	MoveL Offs(p0,158.4466,180.3462, 0), v100, z5, tool0;
	MoveL Offs(p0,157.43040000000002,179.7648, 0), v100, z5, tool0;
	MoveL Offs(p0,156.14780000000002,179.25060000000002, 0), v100, z5, tool0;
	MoveL Offs(p0,154.6,178.8, 0), v100, z5, tool0;
	MoveL Offs(p0,152.49280000000005,178.35360000000009, 0), v100, z5, tool0;
	MoveL Offs(p0,151.33119999999997,178.07639999999998, 0), v100, z5, tool0;
	MoveL Offs(p0,150.12640000000002,177.77280000000002, 0), v100, z5, tool0;
	MoveL Offs(p0,148.9,177.45, 0), v100, z5, tool0;
	MoveL Offs(p0,147.6736,177.11520000000002, 0), v100, z5, tool0;
	MoveL Offs(p0,146.46880000000002,176.7756, 0), v100, z5, tool0;
	MoveL Offs(p0,145.30720000000002,176.43840000000003, 0), v100, z5, tool0;
	MoveL Offs(p0,144.2104,176.1108, 0), v100, z5, tool0;
	MoveL Offs(p0,143.2,175.8, 0), v100, z5, tool0;
	MoveL Offs(p0,140.56640000000002,175.05440000000004, 0), v100, z5, tool0;
	MoveL Offs(p0,139.6846,174.86759999999998, 0), v100, z5, tool0;
	MoveL Offs(p0,139.0752,174.8272, 0), v100, z5, tool0;
	MoveL Offs(p0,138.725,174.95, 0), v100, z5, tool0;
	MoveL Offs(p0,138.6208,175.25279999999998, 0), v100, z5, tool0;
	MoveL Offs(p0,138.7494,175.7524, 0), v100, z5, tool0;
	MoveL Offs(p0,139.0976,176.46560000000002, 0), v100, z5, tool0;
	MoveL Offs(p0,139.6522,177.4092, 0), v100, z5, tool0;
	MoveL Offs(p0,140.4,178.6, 0), v100, z5, tool0;
	MoveL Offs(p0,142.15320000000003,181.3594, 0), v100, z5, tool0;
	MoveL Offs(p0,142.8384,182.4848, 0), v100, z5, tool0;
	MoveL Offs(p0,143.55,183.675, 0), v100, z5, tool0;
	MoveL Offs(p0,144.27360000000002,184.90720000000002, 0), v100, z5, tool0;
	MoveL Offs(p0,144.9948,186.1586, 0), v100, z5, tool0;
	MoveL Offs(p0,145.69920000000002,187.40640000000002, 0), v100, z5, tool0;
	MoveL Offs(p0,146.37240000000003,188.62780000000004, 0), v100, z5, tool0;
	MoveL Offs(p0,147.0,189.8, 0), v100, z5, tool0;
	MoveL Offs(p0,148.70080000000004,193.01120000000006, 0), v100, z5, tool0;
	MoveL Offs(p0,149.3472,194.0768, 0), v100, z5, tool0;
	MoveL Offs(p0,149.9024,194.80160000000004, 0), v100, z5, tool0;
	MoveL Offs(p0,150.4,195.2, 0), v100, z5, tool0;
	MoveL Offs(p0,150.87359999999998,195.28640000000001, 0), v100, z5, tool0;
	MoveL Offs(p0,151.3568,195.0752, 0), v100, z5, tool0;
	MoveL Offs(p0,151.88320000000002,194.5808, 0), v100, z5, tool0;
	MoveL Offs(p0,152.4864,193.8176, 0), v100, z5, tool0;
	MoveL Offs(p0,153.2,192.8, 0), v100, z5, tool0;
	MoveL Offs(p0,155.14880000000002,190.1568, 0), v100, z5, tool0;
	MoveL Offs(p0,155.675,189.475, 0), v100, z5, tool0;
	MoveL Offs(p0,156.1952,188.8112, 0), v100, z5, tool0;
	MoveL Offs(p0,156.6986,188.17860000000002, 0), v100, z5, tool0;
	MoveL Offs(p0,157.17440000000002,187.5904, 0), v100, z5, tool0;
	MoveL Offs(p0,157.6118,187.0598, 0), v100, z5, tool0;
	MoveL Offs(p0,158.0,186.6, 0), v100, z5, tool0;
	MoveL Offs(p0,158.0,186.6, 0), v100, z5, tool0;
	MoveJ Offs(p0,306.0,172.0, 10), v100, z1, tool0;
	MoveL Offs(p0,305.975,169.764, 0), v100, z5, tool0;
	MoveL Offs(p0,305.89600000000013,167.84000000000006, 0), v100, z5, tool0;
	MoveL Offs(p0,305.757,166.20399999999998, 0), v100, z5, tool0;
	MoveL Offs(p0,305.552,164.83200000000002, 0), v100, z5, tool0;
	MoveL Offs(p0,305.275,163.7, 0), v100, z5, tool0;
	MoveL Offs(p0,304.92,162.784, 0), v100, z5, tool0;
	MoveL Offs(p0,304.48100000000005,162.06, 0), v100, z5, tool0;
	MoveL Offs(p0,303.95200000000006,161.504, 0), v100, z5, tool0;
	MoveL Offs(p0,303.327,161.092, 0), v100, z5, tool0;
	MoveL Offs(p0,302.6,160.8, 0), v100, z5, tool0;
	MoveL Offs(p0,299.23699999999997,159.66620000000003, 0), v100, z5, tool0;
	MoveL Offs(p0,295.4720000000001,158.11360000000008, 0), v100, z5, tool0;
	MoveL Offs(p0,291.431,156.2154, 0), v100, z5, tool0;
	MoveL Offs(p0,287.24000000000007,154.0448, 0), v100, z5, tool0;
	MoveL Offs(p0,283.025,151.675, 0), v100, z5, tool0;
	MoveL Offs(p0,278.912,149.17919999999998, 0), v100, z5, tool0;
	MoveL Offs(p0,275.027,146.6306, 0), v100, z5, tool0;
	MoveL Offs(p0,271.496,144.10240000000002, 0), v100, z5, tool0;
	MoveL Offs(p0,268.44500000000005,141.6678, 0), v100, z5, tool0;
	MoveL Offs(p0,266.0,139.4, 0), v100, z5, tool0;
	MoveL Offs(p0,261.7404,134.63479999999998, 0), v100, z5, tool0;
	MoveL Offs(p0,258.56320000000005,130.29440000000002, 0), v100, z5, tool0;
	MoveL Offs(p0,256.4708,126.37159999999999, 0), v100, z5, tool0;
	MoveL Offs(p0,255.46560000000005,122.85920000000003, 0), v100, z5, tool0;
	MoveL Offs(p0,255.55,119.75, 0), v100, z5, tool0;
	MoveL Offs(p0,256.7264,117.0368, 0), v100, z5, tool0;
	MoveL Offs(p0,258.99719999999996,114.71239999999997, 0), v100, z5, tool0;
	MoveL Offs(p0,262.3648,112.76960000000001, 0), v100, z5, tool0;
	MoveL Offs(p0,266.83160000000004,111.20120000000001, 0), v100, z5, tool0;
	MoveL Offs(p0,272.4,110.0, 0), v100, z5, tool0;
	MoveL Offs(p0,275.49280000000005,109.58740000000003, 0), v100, z5, tool0;
	MoveL Offs(p0,278.59040000000005,109.31520000000005, 0), v100, z5, tool0;
	MoveL Offs(p0,281.7815999999999,109.19179999999999, 0), v100, z5, tool0;
	MoveL Offs(p0,285.15520000000004,109.22560000000001, 0), v100, z5, tool0;
	MoveL Offs(p0,288.8,109.425, 0), v100, z5, tool0;
	MoveL Offs(p0,292.8048,109.79839999999999, 0), v100, z5, tool0;
	MoveL Offs(p0,297.2584,110.35419999999999, 0), v100, z5, tool0;
	MoveL Offs(p0,302.2496,111.10080000000002, 0), v100, z5, tool0;
	MoveL Offs(p0,307.8672,112.04659999999998, 0), v100, z5, tool0;
	MoveL Offs(p0,314.2,113.2, 0), v100, z5, tool0;
	MoveL Offs(p0,317.7136000000001,113.63040000000004, 0), v100, z5, tool0;
	MoveL Offs(p0,319.1914,113.54560000000001, 0), v100, z5, tool0;
	MoveL Offs(p0,320.61280000000005,113.18719999999999, 0), v100, z5, tool0;
	MoveL Offs(p0,322.075,112.5, 0), v100, z5, tool0;
	MoveL Offs(p0,323.6752,111.4288, 0), v100, z5, tool0;
	MoveL Offs(p0,325.5106,109.91839999999999, 0), v100, z5, tool0;
	MoveL Offs(p0,327.67840000000007,107.9136, 0), v100, z5, tool0;
	MoveL Offs(p0,330.2758,105.35920000000002, 0), v100, z5, tool0;
	MoveL Offs(p0,333.4,102.2, 0), v100, z5, tool0;
	MoveL Offs(p0,345.2,90.0, 0), v100, z5, tool0;
	MoveL Offs(p0,335.0,90.0, 0), v100, z5, tool0;
	MoveL Offs(p0,331.073,89.83140000000002, 0), v100, z5, tool0;
	MoveL Offs(p0,326.5760000000001,89.34720000000002, 0), v100, z5, tool0;
	MoveL Offs(p0,321.63499999999993,88.5798, 0), v100, z5, tool0;
	MoveL Offs(p0,316.37600000000003,87.56160000000001, 0), v100, z5, tool0;
	MoveL Offs(p0,310.925,86.325, 0), v100, z5, tool0;
	MoveL Offs(p0,305.408,84.90239999999999, 0), v100, z5, tool0;
	MoveL Offs(p0,299.95099999999996,83.3262, 0), v100, z5, tool0;
	MoveL Offs(p0,294.68,81.6288, 0), v100, z5, tool0;
	MoveL Offs(p0,289.721,79.8426, 0), v100, z5, tool0;
	MoveL Offs(p0,285.2,78.0, 0), v100, z5, tool0;
	MoveL Offs(p0,281.60640000000006,76.04320000000003, 0), v100, z5, tool0;
	MoveL Offs(p0,279.6056,74.80679999999998, 0), v100, z5, tool0;
	MoveL Offs(p0,277.5232,73.43360000000001, 0), v100, z5, tool0;
	MoveL Offs(p0,275.4,71.95, 0), v100, z5, tool0;
	MoveL Offs(p0,273.2768,70.38239999999999, 0), v100, z5, tool0;
	MoveL Offs(p0,271.1944,68.7572, 0), v100, z5, tool0;
	MoveL Offs(p0,269.1936,67.1008, 0), v100, z5, tool0;
	MoveL Offs(p0,267.3152,65.4396, 0), v100, z5, tool0;
	MoveL Offs(p0,265.6,63.8, 0), v100, z5, tool0;
	MoveL Offs(p0,256.0,54.2, 0), v100, z5, tool0;
	MoveL Offs(p0,252.0,62.0, 0), v100, z5, tool0;
	MoveL Offs(p0,249.06160000000006,68.46360000000001, 0), v100, z5, tool0;
	MoveL Offs(p0,246.61280000000005,75.40480000000002, 0), v100, z5, tool0;
	MoveL Offs(p0,244.66319999999996,82.6892, 0), v100, z5, tool0;
	MoveL Offs(p0,243.22240000000002,90.1824, 0), v100, z5, tool0;
	MoveL Offs(p0,242.3,97.75, 0), v100, z5, tool0;
	MoveL Offs(p0,241.9056,105.2576, 0), v100, z5, tool0;
	MoveL Offs(p0,242.04879999999997,112.5708, 0), v100, z5, tool0;
	MoveL Offs(p0,242.73920000000004,119.55520000000001, 0), v100, z5, tool0;
	MoveL Offs(p0,243.9864,126.0764, 0), v100, z5, tool0;
	MoveL Offs(p0,245.8,132.0, 0), v100, z5, tool0;
	MoveL Offs(p0,247.3344000000001,135.71680000000003, 0), v100, z5, tool0;
	MoveL Offs(p0,248.23359999999997,137.6952, 0), v100, z5, tool0;
	MoveL Offs(p0,249.19520000000003,139.70239999999998, 0), v100, z5, tool0;
	MoveL Offs(p0,250.2,141.7, 0), v100, z5, tool0;
	MoveL Offs(p0,251.2288,143.64960000000002, 0), v100, z5, tool0;
	MoveL Offs(p0,252.26239999999999,145.51280000000003, 0), v100, z5, tool0;
	MoveL Offs(p0,253.28160000000003,147.2512, 0), v100, z5, tool0;
	MoveL Offs(p0,254.2672,148.8264, 0), v100, z5, tool0;
	MoveL Offs(p0,255.2,150.2, 0), v100, z5, tool0;
	MoveL Offs(p0,258.3632,154.18440000000004, 0), v100, z5, tool0;
	MoveL Offs(p0,262.43360000000007,158.36320000000006, 0), v100, z5, tool0;
	MoveL Offs(p0,267.2024,162.59480000000002, 0), v100, z5, tool0;
	MoveL Offs(p0,272.46080000000006,166.73760000000001, 0), v100, z5, tool0;
	MoveL Offs(p0,278.0,170.65, 0), v100, z5, tool0;
	MoveL Offs(p0,283.6112,174.1904, 0), v100, z5, tool0;
	MoveL Offs(p0,289.0856,177.2172, 0), v100, z5, tool0;
	MoveL Offs(p0,294.2144,179.58880000000002, 0), v100, z5, tool0;
	MoveL Offs(p0,298.7888,181.1636, 0), v100, z5, tool0;
	MoveL Offs(p0,302.6,181.8, 0), v100, z5, tool0;
	MoveL Offs(p0,305.00640000000004,180.79840000000002, 0), v100, z5, tool0;
	MoveL Offs(p0,305.35,180.05, 0), v100, z5, tool0;
	MoveL Offs(p0,305.6096,179.0496, 0), v100, z5, tool0;
	MoveL Offs(p0,305.7948,177.7708, 0), v100, z5, tool0;
	MoveL Offs(p0,305.9152,176.18720000000002, 0), v100, z5, tool0;
	MoveL Offs(p0,305.98040000000003,174.2724, 0), v100, z5, tool0;
	MoveL Offs(p0,306.0,172.0, 0), v100, z5, tool0;
	MoveL Offs(p0,306.0,172.0, 0), v100, z5, tool0;
	MoveJ Offs(p0,510.0,155.6, 10), v100, z1, tool0;
	MoveL Offs(p0,507.53460000000007,145.5334, 0), v100, z5, tool0;
	MoveL Offs(p0,504.22080000000017,136.09920000000005, 0), v100, z5, tool0;
	MoveL Offs(p0,500.06219999999996,127.30579999999998, 0), v100, z5, tool0;
	MoveL Offs(p0,495.06239999999997,119.16160000000002, 0), v100, z5, tool0;
	MoveL Offs(p0,489.225,111.675, 0), v100, z5, tool0;
	MoveL Offs(p0,482.5536,104.85439999999998, 0), v100, z5, tool0;
	MoveL Offs(p0,475.0517999999999,98.7082, 0), v100, z5, tool0;
	MoveL Offs(p0,466.7232,93.24480000000001, 0), v100, z5, tool0;
	MoveL Offs(p0,457.5714,88.4726, 0), v100, z5, tool0;
	MoveL Offs(p0,447.6,84.4, 0), v100, z5, tool0;
	MoveL Offs(p0,443.93160000000006,83.08260000000001, 0), v100, z5, tool0;
	MoveL Offs(p0,440.62080000000014,81.99680000000002, 0), v100, z5, tool0;
	MoveL Offs(p0,437.50919999999996,81.12219999999999, 0), v100, z5, tool0;
	MoveL Offs(p0,434.4384,80.43839999999999, 0), v100, z5, tool0;
	MoveL Offs(p0,431.25,79.925, 0), v100, z5, tool0;
	MoveL Offs(p0,427.7856,79.5616, 0), v100, z5, tool0;
	MoveL Offs(p0,423.88680000000005,79.3278, 0), v100, z5, tool0;
	MoveL Offs(p0,419.39520000000005,79.20320000000001, 0), v100, z5, tool0;
	MoveL Offs(p0,414.15240000000006,79.1674, 0), v100, z5, tool0;
	MoveL Offs(p0,408.0,79.2, 0), v100, z5, tool0;
	MoveL Offs(p0,398.902,79.31840000000001, 0), v100, z5, tool0;
	MoveL Offs(p0,390.9920000000001,79.69120000000002, 0), v100, z5, tool0;
	MoveL Offs(p0,384.186,80.34479999999999, 0), v100, z5, tool0;
	MoveL Offs(p0,378.4,81.3056, 0), v100, z5, tool0;
	MoveL Offs(p0,373.55,82.6, 0), v100, z5, tool0;
	MoveL Offs(p0,369.552,84.2544, 0), v100, z5, tool0;
	MoveL Offs(p0,366.322,86.2952, 0), v100, z5, tool0;
	MoveL Offs(p0,363.776,88.7488, 0), v100, z5, tool0;
	MoveL Offs(p0,361.83000000000004,91.64160000000001, 0), v100, z5, tool0;
	MoveL Offs(p0,360.4,95.0, 0), v100, z5, tool0;
	MoveL Offs(p0,359.1992000000001,100.0506, 0), v100, z5, tool0;
	MoveL Offs(p0,358.80960000000016,105.52480000000003, 0), v100, z5, tool0;
	MoveL Offs(p0,359.1904,111.30619999999999, 0), v100, z5, tool0;
	MoveL Offs(p0,360.3008000000001,117.2784, 0), v100, z5, tool0;
	MoveL Offs(p0,362.1,123.325, 0), v100, z5, tool0;
	MoveL Offs(p0,364.5472,129.32959999999997, 0), v100, z5, tool0;
	MoveL Offs(p0,367.60159999999996,135.17579999999998, 0), v100, z5, tool0;
	MoveL Offs(p0,371.2224,140.74720000000002, 0), v100, z5, tool0;
	MoveL Offs(p0,375.3688,145.9274, 0), v100, z5, tool0;
	MoveL Offs(p0,380.0,150.6, 0), v100, z5, tool0;
	MoveL Offs(p0,383.889,153.90980000000002, 0), v100, z5, tool0;
	MoveL Offs(p0,387.5680000000001,156.65440000000007, 0), v100, z5, tool0;
	MoveL Offs(p0,391.115,158.8566, 0), v100, z5, tool0;
	MoveL Offs(p0,394.60800000000006,160.5392, 0), v100, z5, tool0;
	MoveL Offs(p0,398.125,161.725, 0), v100, z5, tool0;
	MoveL Offs(p0,401.74399999999997,162.4368, 0), v100, z5, tool0;
	MoveL Offs(p0,405.543,162.69740000000002, 0), v100, z5, tool0;
	MoveL Offs(p0,409.6,162.52960000000002, 0), v100, z5, tool0;
	MoveL Offs(p0,413.99300000000005,161.9562, 0), v100, z5, tool0;
	MoveL Offs(p0,418.8,161.0, 0), v100, z5, tool0;
	MoveL Offs(p0,427.9466000000001,159.2384, 0), v100, z5, tool0;
	MoveL Offs(p0,437.39680000000016,158.13920000000002, 0), v100, z5, tool0;
	MoveL Offs(p0,446.98619999999994,157.6808, 0), v100, z5, tool0;
	MoveL Offs(p0,456.55039999999997,157.8416, 0), v100, z5, tool0;
	MoveL Offs(p0,465.925,158.6, 0), v100, z5, tool0;
	MoveL Offs(p0,474.9456,159.9344, 0), v100, z5, tool0;
	MoveL Offs(p0,483.4477999999999,161.82319999999999, 0), v100, z5, tool0;
	MoveL Offs(p0,491.26720000000006,164.2448, 0), v100, z5, tool0;
	MoveL Offs(p0,498.23940000000005,167.1776, 0), v100, z5, tool0;
	MoveL Offs(p0,504.2,170.6, 0), v100, z5, tool0;
	MoveL Offs(p0,507.44640000000015,172.81280000000004, 0), v100, z5, tool0;
	MoveL Offs(p0,508.5956,173.51420000000002, 0), v100, z5, tool0;
	MoveL Offs(p0,509.4832,173.9504, 0), v100, z5, tool0;
	MoveL Offs(p0,510.15,174.125, 0), v100, z5, tool0;
	MoveL Offs(p0,510.63680000000005,174.0416, 0), v100, z5, tool0;
	MoveL Offs(p0,510.9844,173.7038, 0), v100, z5, tool0;
	MoveL Offs(p0,511.23360000000014,173.11520000000002, 0), v100, z5, tool0;
	MoveL Offs(p0,511.4252,172.2794, 0), v100, z5, tool0;
	MoveL Offs(p0,511.6,171.2, 0), v100, z5, tool0;
	MoveL Offs(p0,511.69539999999995,168.0698, 0), v100, z5, tool0;
	MoveL Offs(p0,511.61280000000005,166.60160000000002, 0), v100, z5, tool0;
	MoveL Offs(p0,511.475,164.975, 0), v100, z5, tool0;
	MoveL Offs(p0,511.28319999999997,163.2224, 0), v100, z5, tool0;
	MoveL Offs(p0,511.0386,161.37619999999998, 0), v100, z5, tool0;
	MoveL Offs(p0,510.7424000000001,159.46880000000002, 0), v100, z5, tool0;
	MoveL Offs(p0,510.39580000000007,157.5326, 0), v100, z5, tool0;
	MoveL Offs(p0,510.0,155.6, 0), v100, z5, tool0;
	MoveL Offs(p0,510.0,155.6, 0), v100, z5, tool0;
	MoveJ Offs(p0,181.4,171.0, 10), v100, z1, tool0;
	MoveL Offs(p0,184.04000000000008,170.41920000000005, 0), v100, z5, tool0;
	MoveL Offs(p0,185.57599999999996,169.9848, 0), v100, z5, tool0;
	MoveL Offs(p0,187.208,169.4736, 0), v100, z5, tool0;
	MoveL Offs(p0,188.9,168.9, 0), v100, z5, tool0;
	MoveL Offs(p0,190.616,168.27839999999998, 0), v100, z5, tool0;
	MoveL Offs(p0,192.32,167.6232, 0), v100, z5, tool0;
	MoveL Offs(p0,193.97600000000003,166.9488, 0), v100, z5, tool0;
	MoveL Offs(p0,195.548,166.26960000000003, 0), v100, z5, tool0;
	MoveL Offs(p0,197.0,165.6, 0), v100, z5, tool0;
	MoveL Offs(p0,205.6,161.4, 0), v100, z5, tool0;
	MoveL Offs(p0,194.4,154.6, 0), v100, z5, tool0;
	MoveL Offs(p0,191.1044,152.5704, 0), v100, z5, tool0;
	MoveL Offs(p0,187.83520000000004,150.33920000000003, 0), v100, z5, tool0;
	MoveL Offs(p0,184.6188,147.9328, 0), v100, z5, tool0;
	MoveL Offs(p0,181.48160000000001,145.3776, 0), v100, z5, tool0;
	MoveL Offs(p0,178.45,142.7, 0), v100, z5, tool0;
	MoveL Offs(p0,175.5504,139.92639999999997, 0), v100, z5, tool0;
	MoveL Offs(p0,172.80919999999998,137.08319999999998, 0), v100, z5, tool0;
	MoveL Offs(p0,170.2528,134.1968, 0), v100, z5, tool0;
	MoveL Offs(p0,167.90760000000003,131.29360000000003, 0), v100, z5, tool0;
	MoveL Offs(p0,165.8,128.4, 0), v100, z5, tool0;
	MoveL Offs(p0,164.20960000000002,126.35360000000003, 0), v100, z5, tool0;
	MoveL Offs(p0,163.4834,125.67839999999998, 0), v100, z5, tool0;
	MoveL Offs(p0,162.72480000000002,125.2288, 0), v100, z5, tool0;
	MoveL Offs(p0,161.875,125.0, 0), v100, z5, tool0;
	MoveL Offs(p0,160.8752,124.98719999999999, 0), v100, z5, tool0;
	MoveL Offs(p0,159.6666,125.1856, 0), v100, z5, tool0;
	MoveL Offs(p0,158.1904,125.5904, 0), v100, z5, tool0;
	MoveL Offs(p0,156.38780000000003,126.19680000000001, 0), v100, z5, tool0;
	MoveL Offs(p0,154.2,127.0, 0), v100, z5, tool0;
	MoveL Offs(p0,150.75400000000002,128.0432, 0), v100, z5, tool0;
	MoveL Offs(p0,146.98400000000004,128.88960000000003, 0), v100, z5, tool0;
	MoveL Offs(p0,143.022,129.53439999999998, 0), v100, z5, tool0;
	MoveL Offs(p0,139.0,129.9728, 0), v100, z5, tool0;
	MoveL Offs(p0,135.05,130.2, 0), v100, z5, tool0;
	MoveL Offs(p0,131.304,130.21120000000002, 0), v100, z5, tool0;
	MoveL Offs(p0,127.894,130.0016, 0), v100, z5, tool0;
	MoveL Offs(p0,124.952,129.56640000000002, 0), v100, z5, tool0;
	MoveL Offs(p0,122.61000000000001,128.9008, 0), v100, z5, tool0;
	MoveL Offs(p0,121.0,128.0, 0), v100, z5, tool0;
	MoveL Offs(p0,119.25280000000002,125.62240000000001, 0), v100, z5, tool0;
	MoveL Offs(p0,118.9,124.875, 0), v100, z5, tool0;
	MoveL Offs(p0,118.5952,124.09759999999999, 0), v100, z5, tool0;
	MoveL Offs(p0,118.34560000000002,123.3058, 0), v100, z5, tool0;
	MoveL Offs(p0,118.15840000000003,122.51520000000001, 0), v100, z5, tool0;
	MoveL Offs(p0,118.04080000000002,121.74140000000003, 0), v100, z5, tool0;
	MoveL Offs(p0,118.0,121.0, 0), v100, z5, tool0;
	MoveL Offs(p0,118.41600000000001,118.59380000000002, 0), v100, z5, tool0;
	MoveL Offs(p0,119.60000000000002,115.7664, 0), v100, z5, tool0;
	MoveL Offs(p0,121.45599999999999,112.62460000000002, 0), v100, z5, tool0;
	MoveL Offs(p0,123.888,109.27520000000001, 0), v100, z5, tool0;
	MoveL Offs(p0,126.8,105.825, 0), v100, z5, tool0;
	MoveL Offs(p0,130.096,102.3808, 0), v100, z5, tool0;
	MoveL Offs(p0,133.68,99.0494, 0), v100, z5, tool0;
	MoveL Offs(p0,137.45600000000002,95.9376, 0), v100, z5, tool0;
	MoveL Offs(p0,141.328,93.15220000000002, 0), v100, z5, tool0;
	MoveL Offs(p0,145.2,90.8, 0), v100, z5, tool0;
	MoveL Offs(p0,148.10080000000005,89.01280000000003, 0), v100, z5, tool0;
	MoveL Offs(p0,149.1672,88.12519999999999, 0), v100, z5, tool0;
	MoveL Offs(p0,150.0224,87.1584, 0), v100, z5, tool0;
	MoveL Offs(p0,150.7,86.05, 0), v100, z5, tool0;
	MoveL Offs(p0,151.2336,84.7376, 0), v100, z5, tool0;
	MoveL Offs(p0,151.6568,83.1588, 0), v100, z5, tool0;
	MoveL Offs(p0,152.00320000000002,81.25120000000001, 0), v100, z5, tool0;
	MoveL Offs(p0,152.3064,78.9524, 0), v100, z5, tool0;
	MoveL Offs(p0,152.6,76.2, 0), v100, z5, tool0;
	MoveL Offs(p0,153.02400000000006,72.40480000000002, 0), v100, z5, tool0;
	MoveL Offs(p0,153.27499999999998,70.5012, 0), v100, z5, tool0;
	MoveL Offs(p0,153.544,68.6384, 0), v100, z5, tool0;
	MoveL Offs(p0,153.825,66.85, 0), v100, z5, tool0;
	MoveL Offs(p0,154.11200000000002,65.16959999999999, 0), v100, z5, tool0;
	MoveL Offs(p0,154.399,63.6308, 0), v100, z5, tool0;
	MoveL Offs(p0,154.68,62.2672, 0), v100, z5, tool0;
	MoveL Offs(p0,154.949,61.1124, 0), v100, z5, tool0;
	MoveL Offs(p0,155.2,60.2, 0), v100, z5, tool0;
	MoveL Offs(p0,156.6,55.2, 0), v100, z5, tool0;
	MoveL Offs(p0,150.8,59.2, 0), v100, z5, tool0;
	MoveL Offs(p0,147.62780000000004,61.26780000000001, 0), v100, z5, tool0;
	MoveL Offs(p0,144.26240000000004,63.14240000000002, 0), v100, z5, tool0;
	MoveL Offs(p0,140.7506,64.81060000000001, 0), v100, z5, tool0;
	MoveL Offs(p0,137.13920000000002,66.25919999999999, 0), v100, z5, tool0;
	MoveL Offs(p0,133.475,67.475, 0), v100, z5, tool0;
	MoveL Offs(p0,129.8048,68.44480000000001, 0), v100, z5, tool0;
	MoveL Offs(p0,126.1754,69.1554, 0), v100, z5, tool0;
	MoveL Offs(p0,122.63360000000003,69.59360000000001, 0), v100, z5, tool0;
	MoveL Offs(p0,119.22619999999999,69.7462, 0), v100, z5, tool0;
	MoveL Offs(p0,116.0,69.6, 0), v100, z5, tool0;
	MoveL Offs(p0,106.6,68.6, 0), v100, z5, tool0;
	MoveL Offs(p0,102.0,81.4, 0), v100, z5, tool0;
	MoveL Offs(p0,99.33760000000001,91.1172, 0), v100, z5, tool0;
	MoveL Offs(p0,98.14880000000002,100.96160000000002, 0), v100, z5, tool0;
	MoveL Offs(p0,98.3712,110.77239999999999, 0), v100, z5, tool0;
	MoveL Offs(p0,99.9424,120.38879999999999, 0), v100, z5, tool0;
	MoveL Offs(p0,102.8,129.65, 0), v100, z5, tool0;
	MoveL Offs(p0,106.8816,138.39520000000002, 0), v100, z5, tool0;
	MoveL Offs(p0,112.12480000000001,146.46359999999999, 0), v100, z5, tool0;
	MoveL Offs(p0,118.4672,153.69440000000003, 0), v100, z5, tool0;
	MoveL Offs(p0,125.84639999999999,159.92680000000001, 0), v100, z5, tool0;
	MoveL Offs(p0,134.2,165.0, 0), v100, z5, tool0;
	MoveL Offs(p0,138.71300000000002,167.16060000000002, 0), v100, z5, tool0;
	MoveL Offs(p0,143.16000000000003,168.96480000000003, 0), v100, z5, tool0;
	MoveL Offs(p0,147.583,170.41619999999998, 0), v100, z5, tool0;
	MoveL Offs(p0,152.02400000000003,171.5184, 0), v100, z5, tool0;
	MoveL Offs(p0,156.525,172.275, 0), v100, z5, tool0;
	MoveL Offs(p0,161.128,172.68959999999998, 0), v100, z5, tool0;
	MoveL Offs(p0,165.875,172.76579999999998, 0), v100, z5, tool0;
	MoveL Offs(p0,170.80800000000005,172.5072, 0), v100, z5, tool0;
	MoveL Offs(p0,175.969,171.9174, 0), v100, z5, tool0;
	MoveL Offs(p0,181.4,171.0, 0), v100, z5, tool0;
	MoveL Offs(p0,181.4,171.0, 0), v100, z5, tool0;
	MoveJ Offs(p0,74.6,166.8, 10), v100, z1, tool0;
	MoveL Offs(p0,77.17280000000002,165.32160000000005, 0), v100, z5, tool0;
	MoveL Offs(p0,78.7202,164.32139999999998, 0), v100, z5, tool0;
	MoveL Offs(p0,80.39840000000001,163.18080000000003, 0), v100, z5, tool0;
	MoveL Offs(p0,82.175,161.925, 0), v100, z5, tool0;
	MoveL Offs(p0,84.0176,160.5792, 0), v100, z5, tool0;
	MoveL Offs(p0,85.8938,159.1686, 0), v100, z5, tool0;
	MoveL Offs(p0,87.77120000000001,157.71840000000003, 0), v100, z5, tool0;
	MoveL Offs(p0,89.6174,156.2538, 0), v100, z5, tool0;
	MoveL Offs(p0,91.4,154.8, 0), v100, z5, tool0;
	MoveL Offs(p0,101.6,146.0, 0), v100, z5, tool0;
	MoveL Offs(p0,97.8,136.0, 0), v100, z5, tool0;
	MoveL Offs(p0,96.63680000000002,132.6048, 0), v100, z5, tool0;
	MoveL Offs(p0,96.09719999999999,130.9222, 0), v100, z5, tool0;
	MoveL Offs(p0,95.5984,129.28640000000001, 0), v100, z5, tool0;
	MoveL Offs(p0,95.15,127.725, 0), v100, z5, tool0;
	MoveL Offs(p0,94.7616,126.26559999999999, 0), v100, z5, tool0;
	MoveL Offs(p0,94.4428,124.9358, 0), v100, z5, tool0;
	MoveL Offs(p0,94.20320000000001,123.76320000000001, 0), v100, z5, tool0;
	MoveL Offs(p0,94.0524,122.77540000000002, 0), v100, z5, tool0;
	MoveL Offs(p0,94.0,122.0, 0), v100, z5, tool0;
	MoveL Offs(p0,93.52440000000001,118.99960000000002, 0), v100, z5, tool0;
	MoveL Offs(p0,92.18720000000002,117.48480000000002, 0), v100, z5, tool0;
	MoveL Offs(p0,90.1228,117.34520000000002, 0), v100, z5, tool0;
	MoveL Offs(p0,87.46560000000001,118.4704, 0), v100, z5, tool0;
	MoveL Offs(p0,84.35,120.75, 0), v100, z5, tool0;
	MoveL Offs(p0,80.9104,124.07359999999998, 0), v100, z5, tool0;
	MoveL Offs(p0,77.28119999999998,128.3308, 0), v100, z5, tool0;
	MoveL Offs(p0,73.5968,133.4112, 0), v100, z5, tool0;
	MoveL Offs(p0,69.9916,139.20440000000002, 0), v100, z5, tool0;
	MoveL Offs(p0,66.6,145.6, 0), v100, z5, tool0;
	MoveL Offs(p0,64.8994,149.04300000000003, 0), v100, z5, tool0;
	MoveL Offs(p0,63.50720000000001,151.97600000000006, 0), v100, z5, tool0;
	MoveL Offs(p0,62.407799999999995,154.46499999999997, 0), v100, z5, tool0;
	MoveL Offs(p0,61.5856,156.57600000000002, 0), v100, z5, tool0;
	MoveL Offs(p0,61.025,158.375, 0), v100, z5, tool0;
	MoveL Offs(p0,60.71039999999999,159.92799999999997, 0), v100, z5, tool0;
	MoveL Offs(p0,60.6262,161.30100000000002, 0), v100, z5, tool0;
	MoveL Offs(p0,60.7568,162.56, 0), v100, z5, tool0;
	MoveL Offs(p0,61.0866,163.77100000000002, 0), v100, z5, tool0;
	MoveL Offs(p0,61.6,165.0, 0), v100, z5, tool0;
	MoveL Offs(p0,63.201600000000006,167.83680000000007, 0), v100, z5, tool0;
	MoveL Offs(p0,64.01740000000001,168.7782, 0), v100, z5, tool0;
	MoveL Offs(p0,64.90880000000001,169.40640000000002, 0), v100, z5, tool0;
	MoveL Offs(p0,65.925,169.725, 0), v100, z5, tool0;
	MoveL Offs(p0,67.1152,169.7376, 0), v100, z5, tool0;
	MoveL Offs(p0,68.52860000000001,169.4478, 0), v100, z5, tool0;
	MoveL Offs(p0,70.21440000000001,168.85920000000002, 0), v100, z5, tool0;
	MoveL Offs(p0,72.2218,167.9754, 0), v100, z5, tool0;
	MoveL Offs(p0,74.6,166.8, 0), v100, z5, tool0;
	MoveL Offs(p0,74.6,166.8, 0), v100, z5, tool0;
	MoveJ Offs(p0,247.6,158.2, 10), v100, z1, tool0;
	MoveL Offs(p0,252.2,158.0, 0), v100, z5, tool0;
	MoveL Offs(p0,248.2,152.2, 0), v100, z5, tool0;
	MoveL Offs(p0,246.82720000000012,150.19520000000006, 0), v100, z5, tool0;
	MoveL Offs(p0,246.1228,149.07879999999997, 0), v100, z5, tool0;
	MoveL Offs(p0,245.42560000000003,147.9216, 0), v100, z5, tool0;
	MoveL Offs(p0,244.75,146.75, 0), v100, z5, tool0;
	MoveL Offs(p0,244.11040000000003,145.5904, 0), v100, z5, tool0;
	MoveL Offs(p0,243.5212,144.4692, 0), v100, z5, tool0;
	MoveL Offs(p0,242.99680000000004,143.4128, 0), v100, z5, tool0;
	MoveL Offs(p0,242.5516,142.44760000000002, 0), v100, z5, tool0;
	MoveL Offs(p0,242.2,141.6, 0), v100, z5, tool0;
	MoveL Offs(p0,241.1328000000001,139.28320000000002, 0), v100, z5, tool0;
	MoveL Offs(p0,240.4252,138.4158, 0), v100, z5, tool0;
	MoveL Offs(p0,239.5184,137.7056, 0), v100, z5, tool0;
	MoveL Offs(p0,238.35,137.125, 0), v100, z5, tool0;
	MoveL Offs(p0,236.8576,136.6464, 0), v100, z5, tool0;
	MoveL Offs(p0,234.9788,136.2422, 0), v100, z5, tool0;
	MoveL Offs(p0,232.65120000000007,135.8848, 0), v100, z5, tool0;
	MoveL Offs(p0,229.81239999999997,135.5466, 0), v100, z5, tool0;
	MoveL Offs(p0,226.4,135.2, 0), v100, z5, tool0;
	MoveL Offs(p0,218.27900000000005,133.9028, 0), v100, z5, tool0;
	MoveL Offs(p0,210.36800000000002,131.78240000000002, 0), v100, z5, tool0;
	MoveL Offs(p0,202.865,128.9756, 0), v100, z5, tool0;
	MoveL Offs(p0,195.968,125.61920000000002, 0), v100, z5, tool0;
	MoveL Offs(p0,189.875,121.85, 0), v100, z5, tool0;
	MoveL Offs(p0,184.784,117.8048, 0), v100, z5, tool0;
	MoveL Offs(p0,180.89299999999997,113.62039999999999, 0), v100, z5, tool0;
	MoveL Offs(p0,178.40000000000003,109.4336, 0), v100, z5, tool0;
	MoveL Offs(p0,177.503,105.38119999999999, 0), v100, z5, tool0;
	MoveL Offs(p0,178.4,101.6, 0), v100, z5, tool0;
	MoveL Offs(p0,180.97600000000006,98.31360000000004, 0), v100, z5, tool0;
	MoveL Offs(p0,182.909,96.88040000000001, 0), v100, z5, tool0;
	MoveL Offs(p0,185.32800000000003,95.56480000000002, 0), v100, z5, tool0;
	MoveL Offs(p0,188.275,94.35, 0), v100, z5, tool0;
	MoveL Offs(p0,191.792,93.2192, 0), v100, z5, tool0;
	MoveL Offs(p0,195.921,92.1556, 0), v100, z5, tool0;
	MoveL Offs(p0,200.704,91.14240000000002, 0), v100, z5, tool0;
	MoveL Offs(p0,206.183,90.16279999999999, 0), v100, z5, tool0;
	MoveL Offs(p0,212.4,89.2, 0), v100, z5, tool0;
	MoveL Offs(p0,215.82420000000002,88.67300000000002, 0), v100, z5, tool0;
	MoveL Offs(p0,219.10560000000004,88.17600000000002, 0), v100, z5, tool0;
	MoveL Offs(p0,222.19740000000002,87.71499999999999, 0), v100, z5, tool0;
	MoveL Offs(p0,225.05280000000002,87.296, 0), v100, z5, tool0;
	MoveL Offs(p0,227.625,86.925, 0), v100, z5, tool0;
	MoveL Offs(p0,229.8672,86.608, 0), v100, z5, tool0;
	MoveL Offs(p0,231.7326,86.351, 0), v100, z5, tool0;
	MoveL Offs(p0,233.17440000000002,86.16000000000001, 0), v100, z5, tool0;
	MoveL Offs(p0,234.1458,86.041, 0), v100, z5, tool0;
	MoveL Offs(p0,234.6,86.0, 0), v100, z5, tool0;
	MoveL Offs(p0,235.90240000000003,83.952, 0), v100, z5, tool0;
	MoveL Offs(p0,236.375,82.9, 0), v100, z5, tool0;
	MoveL Offs(p0,236.88959999999997,81.67999999999999, 0), v100, z5, tool0;
	MoveL Offs(p0,237.43779999999998,80.31599999999999, 0), v100, z5, tool0;
	MoveL Offs(p0,238.0112,78.83200000000001, 0), v100, z5, tool0;
	MoveL Offs(p0,238.6014,77.252, 0), v100, z5, tool0;
	MoveL Offs(p0,239.2,75.6, 0), v100, z5, tool0;
	MoveL Offs(p0,240.38080000000005,72.06560000000003, 0), v100, z5, tool0;
	MoveL Offs(p0,241.02519999999998,70.3044, 0), v100, z5, tool0;
	MoveL Offs(p0,241.6864,68.58879999999999, 0), v100, z5, tool0;
	MoveL Offs(p0,242.35,66.95, 0), v100, z5, tool0;
	MoveL Offs(p0,243.00159999999997,65.4192, 0), v100, z5, tool0;
	MoveL Offs(p0,243.62679999999995,64.02759999999999, 0), v100, z5, tool0;
	MoveL Offs(p0,244.21120000000002,62.80640000000001, 0), v100, z5, tool0;
	MoveL Offs(p0,244.74040000000005,61.78679999999999, 0), v100, z5, tool0;
	MoveL Offs(p0,245.2,61.0, 0), v100, z5, tool0;
	MoveL Offs(p0,247.04320000000007,58.04160000000002, 0), v100, z5, tool0;
	MoveL Offs(p0,247.54180000000002,56.9464, 0), v100, z5, tool0;
	MoveL Offs(p0,247.7536,56.100800000000014, 0), v100, z5, tool0;
	MoveL Offs(p0,247.675,55.5, 0), v100, z5, tool0;
	MoveL Offs(p0,247.30239999999998,55.1392, 0), v100, z5, tool0;
	MoveL Offs(p0,246.6322,55.0136, 0), v100, z5, tool0;
	MoveL Offs(p0,245.66080000000002,55.11840000000001, 0), v100, z5, tool0;
	MoveL Offs(p0,244.3846,55.448800000000006, 0), v100, z5, tool0;
	MoveL Offs(p0,242.8,56.0, 0), v100, z5, tool0;
	MoveL Offs(p0,238.1166,57.2124, 0), v100, z5, tool0;
	MoveL Offs(p0,232.18880000000007,57.87520000000002, 0), v100, z5, tool0;
	MoveL Offs(p0,225.32019999999997,58.0268, 0), v100, z5, tool0;
	MoveL Offs(p0,217.81440000000006,57.705600000000004, 0), v100, z5, tool0;
	MoveL Offs(p0,209.975,56.95, 0), v100, z5, tool0;
	MoveL Offs(p0,202.10559999999998,55.798399999999994, 0), v100, z5, tool0;
	MoveL Offs(p0,194.50979999999998,54.28920000000001, 0), v100, z5, tool0;
	MoveL Offs(p0,187.49120000000002,52.46079999999999, 0), v100, z5, tool0;
	MoveL Offs(p0,181.35340000000002,50.351600000000005, 0), v100, z5, tool0;
	MoveL Offs(p0,176.4,48.0, 0), v100, z5, tool0;
	MoveL Offs(p0,174.28800000000007,46.739200000000004, 0), v100, z5, tool0;
	MoveL Offs(p0,173.29500000000002,46.1658, 0), v100, z5, tool0;
	MoveL Offs(p0,172.368,45.641600000000004, 0), v100, z5, tool0;
	MoveL Offs(p0,171.525,45.175, 0), v100, z5, tool0;
	MoveL Offs(p0,170.78400000000002,44.7744, 0), v100, z5, tool0;
	MoveL Offs(p0,170.163,44.4482, 0), v100, z5, tool0;
	MoveL Offs(p0,169.68,44.2048, 0), v100, z5, tool0;
	MoveL Offs(p0,169.353,44.0526, 0), v100, z5, tool0;
	MoveL Offs(p0,169.2,44.0, 0), v100, z5, tool0;
	MoveL Offs(p0,166.80419999999998,48.066199999999995, 0), v100, z5, tool0;
	MoveL Offs(p0,165.7184,50.8224, 0), v100, z5, tool0;
	MoveL Offs(p0,164.575,54.025, 0), v100, z5, tool0;
	MoveL Offs(p0,163.42559999999997,57.5216, 0), v100, z5, tool0;
	MoveL Offs(p0,162.3218,61.159800000000004, 0), v100, z5, tool0;
	MoveL Offs(p0,161.3152,64.78720000000001, 0), v100, z5, tool0;
	MoveL Offs(p0,160.4574,68.25140000000002, 0), v100, z5, tool0;
	MoveL Offs(p0,159.8,71.4, 0), v100, z5, tool0;
	MoveL Offs(p0,159.24020000000002,75.45660000000001, 0), v100, z5, tool0;
	MoveL Offs(p0,158.99360000000004,79.78080000000003, 0), v100, z5, tool0;
	MoveL Offs(p0,159.0494,84.30420000000001, 0), v100, z5, tool0;
	MoveL Offs(p0,159.3968,88.95840000000003, 0), v100, z5, tool0;
	MoveL Offs(p0,160.025,93.675, 0), v100, z5, tool0;
	MoveL Offs(p0,160.9232,98.3856, 0), v100, z5, tool0;
	MoveL Offs(p0,162.0806,103.02179999999998, 0), v100, z5, tool0;
	MoveL Offs(p0,163.4864,107.51520000000001, 0), v100, z5, tool0;
	MoveL Offs(p0,165.1298,111.79740000000001, 0), v100, z5, tool0;
	MoveL Offs(p0,167.0,115.8, 0), v100, z5, tool0;
	MoveL Offs(p0,169.18,119.63700000000001, 0), v100, z5, tool0;
	MoveL Offs(p0,171.93600000000006,123.64800000000002, 0), v100, z5, tool0;
	MoveL Offs(p0,175.17199999999997,127.74299999999998, 0), v100, z5, tool0;
	MoveL Offs(p0,178.792,131.83200000000002, 0), v100, z5, tool0;
	MoveL Offs(p0,182.7,135.825, 0), v100, z5, tool0;
	MoveL Offs(p0,186.8,139.632, 0), v100, z5, tool0;
	MoveL Offs(p0,190.996,143.163, 0), v100, z5, tool0;
	MoveL Offs(p0,195.192,146.32800000000003, 0), v100, z5, tool0;
	MoveL Offs(p0,199.292,149.03699999999998, 0), v100, z5, tool0;
	MoveL Offs(p0,203.2,151.2, 0), v100, z5, tool0;
	MoveL Offs(p0,206.5072,152.7036, 0), v100, z5, tool0;
	MoveL Offs(p0,210.02560000000008,154.08480000000003, 0), v100, z5, tool0;
	MoveL Offs(p0,213.6904,155.32920000000001, 0), v100, z5, tool0;
	MoveL Offs(p0,217.43680000000003,156.42239999999998, 0), v100, z5, tool0;
	MoveL Offs(p0,221.2,157.35, 0), v100, z5, tool0;
	MoveL Offs(p0,224.9152,158.0976, 0), v100, z5, tool0;
	MoveL Offs(p0,228.5176,158.6508, 0), v100, z5, tool0;
	MoveL Offs(p0,231.94240000000005,158.9952, 0), v100, z5, tool0;
	MoveL Offs(p0,235.1248,159.11640000000003, 0), v100, z5, tool0;
	MoveL Offs(p0,238.0,159.0, 0), v100, z5, tool0;
	MoveL Offs(p0,240.817,158.68859999999998, 0), v100, z5, tool0;
	MoveL Offs(p0,241.84,158.60320000000002, 0), v100, z5, tool0;
	MoveL Offs(p0,242.875,158.525, 0), v100, z5, tool0;
	MoveL Offs(p0,243.904,158.4528, 0), v100, z5, tool0;
	MoveL Offs(p0,244.90900000000002,158.38539999999998, 0), v100, z5, tool0;
	MoveL Offs(p0,245.872,158.32160000000002, 0), v100, z5, tool0;
	MoveL Offs(p0,246.775,158.2602, 0), v100, z5, tool0;
	MoveL Offs(p0,247.6,158.2, 0), v100, z5, tool0;
	MoveL Offs(p0,247.6,158.2, 0), v100, z5, tool0;
	MoveJ Offs(p0,316.6,127.2, 10), v100, z1, tool0;
	MoveL Offs(p0,317.69760000000014,124.67520000000002, 0), v100, z5, tool0;
	MoveL Offs(p0,318.1624,123.52079999999998, 0), v100, z5, tool0;
	MoveL Offs(p0,318.5648,122.4576, 0), v100, z5, tool0;
	MoveL Offs(p0,318.9,121.5, 0), v100, z5, tool0;
	MoveL Offs(p0,319.1632,120.6624, 0), v100, z5, tool0;
	MoveL Offs(p0,319.3496,119.95920000000001, 0), v100, z5, tool0;
	MoveL Offs(p0,319.4544,119.40480000000002, 0), v100, z5, tool0;
	MoveL Offs(p0,319.4728,119.0136, 0), v100, z5, tool0;
	MoveL Offs(p0,319.4,118.8, 0), v100, z5, tool0;
	MoveL Offs(p0,315.29600000000005,117.70880000000004, 0), v100, z5, tool0;
	MoveL Offs(p0,311.183,116.89020000000001, 0), v100, z5, tool0;
	MoveL Offs(p0,306.2,115.97440000000002, 0), v100, z5, tool0;
	MoveL Offs(p0,300.725,115.025, 0), v100, z5, tool0;
	MoveL Offs(p0,295.13599999999997,114.10559999999998, 0), v100, z5, tool0;
	MoveL Offs(p0,289.811,113.2798, 0), v100, z5, tool0;
	MoveL Offs(p0,285.12800000000004,112.61120000000001, 0), v100, z5, tool0;
	MoveL Offs(p0,281.46500000000003,112.1634, 0), v100, z5, tool0;
	MoveL Offs(p0,279.2,112.0, 0), v100, z5, tool0;
	MoveL Offs(p0,276.77700000000004,112.1152, 0), v100, z5, tool0;
	MoveL Offs(p0,274.24000000000007,112.44160000000004, 0), v100, z5, tool0;
	MoveL Offs(p0,271.667,112.95039999999999, 0), v100, z5, tool0;
	MoveL Offs(p0,269.136,113.61280000000002, 0), v100, z5, tool0;
	MoveL Offs(p0,266.725,114.4, 0), v100, z5, tool0;
	MoveL Offs(p0,264.512,115.28320000000001, 0), v100, z5, tool0;
	MoveL Offs(p0,262.575,116.2336, 0), v100, z5, tool0;
	MoveL Offs(p0,260.992,117.22240000000002, 0), v100, z5, tool0;
	MoveL Offs(p0,259.841,118.22080000000001, 0), v100, z5, tool0;
	MoveL Offs(p0,259.2,119.2, 0), v100, z5, tool0;
	MoveL Offs(p0,258.98260000000005,122.45520000000002, 0), v100, z5, tool0;
	MoveL Offs(p0,260.34080000000006,126.32960000000006, 0), v100, z5, tool0;
	MoveL Offs(p0,263.0502,130.62640000000002, 0), v100, z5, tool0;
	MoveL Offs(p0,266.8864,135.1488, 0), v100, z5, tool0;
	MoveL Offs(p0,271.625,139.7, 0), v100, z5, tool0;
	MoveL Offs(p0,277.0416,144.08319999999998, 0), v100, z5, tool0;
	MoveL Offs(p0,282.9118,148.10160000000002, 0), v100, z5, tool0;
	MoveL Offs(p0,289.01120000000003,151.55840000000003, 0), v100, z5, tool0;
	MoveL Offs(p0,295.1154,154.25680000000003, 0), v100, z5, tool0;
	MoveL Offs(p0,301.0,156.0, 0), v100, z5, tool0;
	MoveL Offs(p0,303.8768000000001,156.47680000000005, 0), v100, z5, tool0;
	MoveL Offs(p0,304.94019999999995,156.44819999999999, 0), v100, z5, tool0;
	MoveL Offs(p0,305.8224,156.1664, 0), v100, z5, tool0;
	MoveL Offs(p0,306.575,155.575, 0), v100, z5, tool0;
	MoveL Offs(p0,307.2496,154.61759999999998, 0), v100, z5, tool0;
	MoveL Offs(p0,307.8978,153.23780000000002, 0), v100, z5, tool0;
	MoveL Offs(p0,308.57120000000003,151.37920000000003, 0), v100, z5, tool0;
	MoveL Offs(p0,309.3214,148.9854, 0), v100, z5, tool0;
	MoveL Offs(p0,310.2,146.0, 0), v100, z5, tool0;
	MoveL Offs(p0,311.3840000000001,142.14400000000003, 0), v100, z5, tool0;
	MoveL Offs(p0,312.036,140.087, 0), v100, z5, tool0;
	MoveL Offs(p0,312.71200000000005,138.0, 0), v100, z5, tool0;
	MoveL Offs(p0,313.4,135.925, 0), v100, z5, tool0;
	MoveL Offs(p0,314.08799999999997,133.904, 0), v100, z5, tool0;
	MoveL Offs(p0,314.764,131.97899999999998, 0), v100, z5, tool0;
	MoveL Offs(p0,315.41600000000005,130.192, 0), v100, z5, tool0;
	MoveL Offs(p0,316.03200000000004,128.585, 0), v100, z5, tool0;
	MoveL Offs(p0,316.6,127.2, 0), v100, z5, tool0;
	MoveL Offs(p0,316.6,127.2, 0), v100, z5, tool0;
	MoveJ Offs(p0,236.8,132.8, 10), v100, z1, tool0;
	MoveL Offs(p0,238.77280000000002,130.28, 0), v100, z5, tool0;
	MoveL Offs(p0,238.7054,129.552, 0), v100, z5, tool0;
	MoveL Offs(p0,238.52160000000003,128.704, 0), v100, z5, tool0;
	MoveL Offs(p0,238.22020000000003,127.724, 0), v100, z5, tool0;
	MoveL Offs(p0,237.8,126.6, 0), v100, z5, tool0;
	MoveL Offs(p0,237.22880000000004,124.26240000000004, 0), v100, z5, tool0;
	MoveL Offs(p0,236.97020000000003,122.5806, 0), v100, z5, tool0;
	MoveL Offs(p0,236.7344,120.6192, 0), v100, z5, tool0;
	MoveL Offs(p0,236.525,118.425, 0), v100, z5, tool0;
	MoveL Offs(p0,236.34560000000002,116.04479999999998, 0), v100, z5, tool0;
	MoveL Offs(p0,236.1998,113.52539999999999, 0), v100, z5, tool0;
	MoveL Offs(p0,236.09120000000001,110.9136, 0), v100, z5, tool0;
	MoveL Offs(p0,236.02340000000004,108.25619999999999, 0), v100, z5, tool0;
	MoveL Offs(p0,236.0,105.6, 0), v100, z5, tool0;
	MoveL Offs(p0,236.0,89.6, 0), v100, z5, tool0;
	MoveL Offs(p0,229.6,90.6, 0), v100, z5, tool0;
	MoveL Offs(p0,226.9168000000001,91.02240000000003, 0), v100, z5, tool0;
	MoveL Offs(p0,225.24219999999997,91.2696, 0), v100, z5, tool0;
	MoveL Offs(p0,223.39840000000004,91.53120000000001, 0), v100, z5, tool0;
	MoveL Offs(p0,221.425,91.8, 0), v100, z5, tool0;
	MoveL Offs(p0,219.3616,92.06880000000001, 0), v100, z5, tool0;
	MoveL Offs(p0,217.2478,92.33039999999998, 0), v100, z5, tool0;
	MoveL Offs(p0,215.1232,92.5776, 0), v100, z5, tool0;
	MoveL Offs(p0,213.02740000000003,92.80320000000002, 0), v100, z5, tool0;
	MoveL Offs(p0,211.0,93.0, 0), v100, z5, tool0;
	MoveL Offs(p0,201.3376,94.36460000000002, 0), v100, z5, tool0;
	MoveL Offs(p0,193.48480000000004,96.26080000000003, 0), v100, z5, tool0;
	MoveL Offs(p0,187.46319999999997,98.6322, 0), v100, z5, tool0;
	MoveL Offs(p0,183.29440000000005,101.4224, 0), v100, z5, tool0;
	MoveL Offs(p0,181.0,104.575, 0), v100, z5, tool0;
	MoveL Offs(p0,180.60160000000002,108.0336, 0), v100, z5, tool0;
	MoveL Offs(p0,182.1208,111.74180000000001, 0), v100, z5, tool0;
	MoveL Offs(p0,185.57920000000001,115.64320000000002, 0), v100, z5, tool0;
	MoveL Offs(p0,190.9984,119.68140000000001, 0), v100, z5, tool0;
	MoveL Offs(p0,198.4,123.8, 0), v100, z5, tool0;
	MoveL Offs(p0,200.57080000000002,124.8232, 0), v100, z5, tool0;
	MoveL Offs(p0,202.85440000000003,125.84160000000004, 0), v100, z5, tool0;
	MoveL Offs(p0,205.2076,126.83840000000001, 0), v100, z5, tool0;
	MoveL Offs(p0,207.58720000000002,127.7968, 0), v100, z5, tool0;
	MoveL Offs(p0,209.95,128.7, 0), v100, z5, tool0;
	MoveL Offs(p0,212.25279999999998,129.5312, 0), v100, z5, tool0;
	MoveL Offs(p0,214.45239999999998,130.2736, 0), v100, z5, tool0;
	MoveL Offs(p0,216.50560000000004,130.9104, 0), v100, z5, tool0;
	MoveL Offs(p0,218.3692,131.4248, 0), v100, z5, tool0;
	MoveL Offs(p0,220.0,131.8, 0), v100, z5, tool0;
	MoveL Offs(p0,223.2406,132.449, 0), v100, z5, tool0;
	MoveL Offs(p0,225.9328000000001,132.96000000000004, 0), v100, z5, tool0;
	MoveL Offs(p0,228.1522,133.339, 0), v100, z5, tool0;
	MoveL Offs(p0,229.9744,133.592, 0), v100, z5, tool0;
	MoveL Offs(p0,231.475,133.725, 0), v100, z5, tool0;
	MoveL Offs(p0,232.72960000000003,133.744, 0), v100, z5, tool0;
	MoveL Offs(p0,233.8138,133.655, 0), v100, z5, tool0;
	MoveL Offs(p0,234.8032,133.464, 0), v100, z5, tool0;
	MoveL Offs(p0,235.77339999999998,133.177, 0), v100, z5, tool0;
	MoveL Offs(p0,236.8,132.8, 0), v100, z5, tool0;
	MoveL Offs(p0,236.8,132.8, 0), v100, z5, tool0;
	MoveJ Offs(p0,154.4,123.4, 10), v100, z1, tool0;
	MoveL Offs(p0,161.8,120.4, 0), v100, z5, tool0;
	MoveL Offs(p0,157.8,110.2, 0), v100, z5, tool0;
	MoveL Offs(p0,156.63680000000002,106.78400000000003, 0), v100, z5, tool0;
	MoveL Offs(p0,156.0972,105.079, 0), v100, z5, tool0;
	MoveL Offs(p0,155.5984,103.41600000000001, 0), v100, z5, tool0;
	MoveL Offs(p0,155.15,101.825, 0), v100, z5, tool0;
	MoveL Offs(p0,154.7616,100.336, 0), v100, z5, tool0;
	MoveL Offs(p0,154.44279999999998,98.979, 0), v100, z5, tool0;
	MoveL Offs(p0,154.2032,97.784, 0), v100, z5, tool0;
	MoveL Offs(p0,154.05239999999998,96.78100000000002, 0), v100, z5, tool0;
	MoveL Offs(p0,154.0,96.0, 0), v100, z5, tool0;
	MoveL Offs(p0,153.55040000000002,93.45760000000003, 0), v100, z5, tool0;
	MoveL Offs(p0,152.96859999999998,92.7114, 0), v100, z5, tool0;
	MoveL Offs(p0,152.1312,92.3168, 0), v100, z5, tool0;
	MoveL Offs(p0,151.025,92.275, 0), v100, z5, tool0;
	MoveL Offs(p0,149.6368,92.5872, 0), v100, z5, tool0;
	MoveL Offs(p0,147.95340000000002,93.25460000000001, 0), v100, z5, tool0;
	MoveL Offs(p0,145.96160000000003,94.2784, 0), v100, z5, tool0;
	MoveL Offs(p0,143.6482,95.65979999999999, 0), v100, z5, tool0;
	MoveL Offs(p0,141.0,97.4, 0), v100, z5, tool0;
	MoveL Offs(p0,136.74640000000002,100.4204, 0), v100, z5, tool0;
	MoveL Offs(p0,132.89120000000003,103.56320000000002, 0), v100, z5, tool0;
	MoveL Offs(p0,129.4728,106.77080000000001, 0), v100, z5, tool0;
	MoveL Offs(p0,126.5296,109.9856, 0), v100, z5, tool0;
	MoveL Offs(p0,124.1,113.15, 0), v100, z5, tool0;
	MoveL Offs(p0,122.2224,116.2064, 0), v100, z5, tool0;
	MoveL Offs(p0,120.93519999999998,119.09720000000002, 0), v100, z5, tool0;
	MoveL Offs(p0,120.27680000000001,121.76480000000001, 0), v100, z5, tool0;
	MoveL Offs(p0,120.28560000000002,124.1516, 0), v100, z5, tool0;
	MoveL Offs(p0,121.0,126.2, 0), v100, z5, tool0;
	MoveL Offs(p0,124.30080000000002,127.46400000000006, 0), v100, z5, tool0;
	MoveL Offs(p0,127.2442,127.71199999999999, 0), v100, z5, tool0;
	MoveL Offs(p0,130.79840000000002,127.72000000000003, 0), v100, z5, tool0;
	MoveL Offs(p0,134.775,127.5, 0), v100, z5, tool0;
	MoveL Offs(p0,138.9856,127.064, 0), v100, z5, tool0;
	MoveL Offs(p0,143.2418,126.424, 0), v100, z5, tool0;
	MoveL Offs(p0,147.35520000000002,125.59200000000001, 0), v100, z5, tool0;
	MoveL Offs(p0,151.1374,124.58000000000001, 0), v100, z5, tool0;
	MoveL Offs(p0,154.4,123.4, 0), v100, z5, tool0;
	MoveL Offs(p0,154.4,123.4, 0), v100, z5, tool0;
	MoveJ Offs(p0,368.6,80.0, 10), v100, z1, tool0;
	MoveL Offs(p0,374.8776000000001,77.93640000000002, 0), v100, z5, tool0;
	MoveL Offs(p0,381.21280000000013,76.18720000000003, 0), v100, z5, tool0;
	MoveL Offs(p0,387.5792,74.7548, 0), v100, z5, tool0;
	MoveL Offs(p0,393.95040000000006,73.6416, 0), v100, z5, tool0;
	MoveL Offs(p0,400.3,72.85, 0), v100, z5, tool0;
	MoveL Offs(p0,406.60159999999996,72.3824, 0), v100, z5, tool0;
	MoveL Offs(p0,412.82879999999994,72.2412, 0), v100, z5, tool0;
	MoveL Offs(p0,418.95520000000005,72.4288, 0), v100, z5, tool0;
	MoveL Offs(p0,424.95439999999996,72.9476, 0), v100, z5, tool0;
	MoveL Offs(p0,430.8,73.8, 0), v100, z5, tool0;
	MoveL Offs(p0,433.03920000000016,74.1958, 0), v100, z5, tool0;
	MoveL Offs(p0,435.1776000000001,74.54240000000003, 0), v100, z5, tool0;
	MoveL Offs(p0,437.18639999999994,74.83860000000001, 0), v100, z5, tool0;
	MoveL Offs(p0,439.0368,75.0832, 0), v100, z5, tool0;
	MoveL Offs(p0,440.7,75.275, 0), v100, z5, tool0;
	MoveL Offs(p0,442.1472,75.41279999999999, 0), v100, z5, tool0;
	MoveL Offs(p0,443.3496,75.49539999999999, 0), v100, z5, tool0;
	MoveL Offs(p0,444.2784,75.5216, 0), v100, z5, tool0;
	MoveL Offs(p0,444.90479999999997,75.4902, 0), v100, z5, tool0;
	MoveL Offs(p0,445.2,75.4, 0), v100, z5, tool0;
	MoveL Offs(p0,443.9728000000002,71.90880000000001, 0), v100, z5, tool0;
	MoveL Offs(p0,441.8322,68.78320000000001, 0), v100, z5, tool0;
	MoveL Offs(p0,438.9344,65.0384, 0), v100, z5, tool0;
	MoveL Offs(p0,435.475,60.9, 0), v100, z5, tool0;
	MoveL Offs(p0,431.6496,56.593599999999995, 0), v100, z5, tool0;
	MoveL Offs(p0,427.65379999999993,52.344799999999985, 0), v100, z5, tool0;
	MoveL Offs(p0,423.68320000000006,48.379200000000004, 0), v100, z5, tool0;
	MoveL Offs(p0,419.93340000000006,44.922399999999996, 0), v100, z5, tool0;
	MoveL Offs(p0,416.6,42.2, 0), v100, z5, tool0;
	MoveL Offs(p0,403.6772000000001,33.536, 0), v100, z5, tool0;
	MoveL Offs(p0,390.04160000000013,26.288000000000004, 0), v100, z5, tool0;
	MoveL Offs(p0,375.9524,20.491999999999997, 0), v100, z5, tool0;
	MoveL Offs(p0,361.66880000000003,16.184, 0), v100, z5, tool0;
	MoveL Offs(p0,347.45,13.4, 0), v100, z5, tool0;
	MoveL Offs(p0,333.5552,12.176, 0), v100, z5, tool0;
	MoveL Offs(p0,320.2436,12.548, 0), v100, z5, tool0;
	MoveL Offs(p0,307.7744,14.552000000000001, 0), v100, z5, tool0;
	MoveL Offs(p0,296.40680000000003,18.224, 0), v100, z5, tool0;
	MoveL Offs(p0,286.4,23.6, 0), v100, z5, tool0;
	MoveL Offs(p0,282.55780000000004,26.2654, 0), v100, z5, tool0;
	MoveL Offs(p0,278.8704000000001,29.05920000000001, 0), v100, z5, tool0;
	MoveL Offs(p0,275.3966,31.9178, 0), v100, z5, tool0;
	MoveL Offs(p0,272.1952,34.7776, 0), v100, z5, tool0;
	MoveL Offs(p0,269.325,37.575, 0), v100, z5, tool0;
	MoveL Offs(p0,266.84479999999996,40.2464, 0), v100, z5, tool0;
	MoveL Offs(p0,264.8134,42.7282, 0), v100, z5, tool0;
	MoveL Offs(p0,263.2896,44.9568, 0), v100, z5, tool0;
	MoveL Offs(p0,262.3322,46.8686, 0), v100, z5, tool0;
	MoveL Offs(p0,262.0,48.4, 0), v100, z5, tool0;
	MoveL Offs(p0,263.21200000000005,53.5188, 0), v100, z5, tool0;
	MoveL Offs(p0,266.65600000000006,58.702400000000026, 0), v100, z5, tool0;
	MoveL Offs(p0,272.044,63.81160000000001, 0), v100, z5, tool0;
	MoveL Offs(p0,279.088,68.70720000000001, 0), v100, z5, tool0;
	MoveL Offs(p0,287.5,73.25, 0), v100, z5, tool0;
	MoveL Offs(p0,296.992,77.30080000000001, 0), v100, z5, tool0;
	MoveL Offs(p0,307.276,80.7204, 0), v100, z5, tool0;
	MoveL Offs(p0,318.064,83.36960000000002, 0), v100, z5, tool0;
	MoveL Offs(p0,329.06800000000004,85.10920000000002, 0), v100, z5, tool0;
	MoveL Offs(p0,340.0,85.8, 0), v100, z5, tool0;
	MoveL Offs(p0,342.32900000000006,85.7942, 0), v100, z5, tool0;
	MoveL Offs(p0,344.7600000000001,85.65760000000003, 0), v100, z5, tool0;
	MoveL Offs(p0,347.299,85.39139999999999, 0), v100, z5, tool0;
	MoveL Offs(p0,349.952,84.99680000000001, 0), v100, z5, tool0;
	MoveL Offs(p0,352.725,84.475, 0), v100, z5, tool0;
	MoveL Offs(p0,355.62399999999997,83.82719999999999, 0), v100, z5, tool0;
	MoveL Offs(p0,358.655,83.05460000000001, 0), v100, z5, tool0;
	MoveL Offs(p0,361.824,82.1584, 0), v100, z5, tool0;
	MoveL Offs(p0,365.13700000000006,81.13980000000001, 0), v100, z5, tool0;
	MoveL Offs(p0,368.6,80.0, 0), v100, z5, tool0;
	MoveL Offs(p0,368.6,80.0, 0), v100, z5, tool0;
	MoveJ Offs(p0,134.4,62.6, 10), v100, z1, tool0;
	MoveL Offs(p0,138.596,60.890400000000014, 0), v100, z5, tool0;
	MoveL Offs(p0,142.45600000000005,59.09920000000002, 0), v100, z5, tool0;
	MoveL Offs(p0,146.028,57.1928, 0), v100, z5, tool0;
	MoveL Offs(p0,149.36,55.1376, 0), v100, z5, tool0;
	MoveL Offs(p0,152.5,52.9, 0), v100, z5, tool0;
	MoveL Offs(p0,155.496,50.4464, 0), v100, z5, tool0;
	MoveL Offs(p0,158.39600000000002,47.7432, 0), v100, z5, tool0;
	MoveL Offs(p0,161.248,44.756800000000005, 0), v100, z5, tool0;
	MoveL Offs(p0,164.1,41.4536, 0), v100, z5, tool0;
	MoveL Offs(p0,167.0,37.8, 0), v100, z5, tool0;
	MoveL Offs(p0,176.6,25.6, 0), v100, z5, tool0;
	MoveL Offs(p0,169.8,26.8, 0), v100, z5, tool0;
	MoveL Offs(p0,165.6394,27.912799999999997, 0), v100, z5, tool0;
	MoveL Offs(p0,160.63520000000005,29.726400000000005, 0), v100, z5, tool0;
	MoveL Offs(p0,155.0238,32.1136, 0), v100, z5, tool0;
	MoveL Offs(p0,149.04160000000002,34.947199999999995, 0), v100, z5, tool0;
	MoveL Offs(p0,142.925,38.1, 0), v100, z5, tool0;
	MoveL Offs(p0,136.9104,41.4448, 0), v100, z5, tool0;
	MoveL Offs(p0,131.23420000000002,44.8544, 0), v100, z5, tool0;
	MoveL Offs(p0,126.13280000000002,48.201600000000006, 0), v100, z5, tool0;
	MoveL Offs(p0,121.84260000000002,51.35920000000001, 0), v100, z5, tool0;
	MoveL Offs(p0,118.6,54.2, 0), v100, z5, tool0;
	MoveL Offs(p0,115.92960000000002,56.929600000000015, 0), v100, z5, tool0;
	MoveL Offs(p0,114.77140000000001,58.2374, 0), v100, z5, tool0;
	MoveL Offs(p0,113.74880000000003,59.476800000000004, 0), v100, z5, tool0;
	MoveL Offs(p0,112.875,60.625, 0), v100, z5, tool0;
	MoveL Offs(p0,112.1632,61.65920000000001, 0), v100, z5, tool0;
	MoveL Offs(p0,111.62660000000001,62.55659999999999, 0), v100, z5, tool0;
	MoveL Offs(p0,111.2784,63.29440000000001, 0), v100, z5, tool0;
	MoveL Offs(p0,111.13180000000003,63.8498, 0), v100, z5, tool0;
	MoveL Offs(p0,111.2,64.2, 0), v100, z5, tool0;
	MoveL Offs(p0,113.44000000000003,65.53120000000003, 0), v100, z5, tool0;
	MoveL Offs(p0,115.304,65.8578, 0), v100, z5, tool0;
	MoveL Offs(p0,117.55200000000002,65.9696, 0), v100, z5, tool0;
	MoveL Offs(p0,120.1,65.875, 0), v100, z5, tool0;
	MoveL Offs(p0,122.86399999999999,65.5824, 0), v100, z5, tool0;
	MoveL Offs(p0,125.76000000000002,65.1002, 0), v100, z5, tool0;
	MoveL Offs(p0,128.704,64.4368, 0), v100, z5, tool0;
	MoveL Offs(p0,131.612,63.60060000000001, 0), v100, z5, tool0;
	MoveL Offs(p0,134.4,62.6, 0), v100, z5, tool0;
	MoveL Offs(p0,134.4,62.6, 0), v100, z5, tool0;
	MoveJ Offs(p0,245.6,49.0, 10), v100, z1, tool0;
	MoveL Offs(p0,248.48160000000007,47.475200000000015, 0), v100, z5, tool0;
	MoveL Offs(p0,250.14139999999998,46.4188, 0), v100, z5, tool0;
	MoveL Offs(p0,251.90080000000003,45.201600000000006, 0), v100, z5, tool0;
	MoveL Offs(p0,253.725,43.85, 0), v100, z5, tool0;
	MoveL Offs(p0,255.5792,42.39039999999999, 0), v100, z5, tool0;
	MoveL Offs(p0,257.4286,40.849199999999996, 0), v100, z5, tool0;
	MoveL Offs(p0,259.2384,39.2528, 0), v100, z5, tool0;
	MoveL Offs(p0,260.97380000000004,37.62760000000001, 0), v100, z5, tool0;
	MoveL Offs(p0,262.6,36.0, 0), v100, z5, tool0;
	MoveL Offs(p0,266.02080000000007,32.544000000000004, 0), v100, z5, tool0;
	MoveL Offs(p0,267.9802,30.708000000000006, 0), v100, z5, tool0;
	MoveL Offs(p0,270.04640000000006,28.848000000000003, 0), v100, z5, tool0;
	MoveL Offs(p0,272.175,27.0, 0), v100, z5, tool0;
	MoveL Offs(p0,274.32160000000005,25.2, 0), v100, z5, tool0;
	MoveL Offs(p0,276.4418,23.484, 0), v100, z5, tool0;
	MoveL Offs(p0,278.49120000000005,21.888, 0), v100, z5, tool0;
	MoveL Offs(p0,280.42539999999997,20.448, 0), v100, z5, tool0;
	MoveL Offs(p0,282.2,19.2, 0), v100, z5, tool0;
	MoveL Offs(p0,285.7936000000001,16.659200000000006, 0), v100, z5, tool0;
	MoveL Offs(p0,287.2184,15.556799999999996, 0), v100, z5, tool0;
	MoveL Offs(p0,288.38880000000006,14.569600000000003, 0), v100, z5, tool0;
	MoveL Offs(p0,289.3,13.7, 0), v100, z5, tool0;
	MoveL Offs(p0,289.9472,12.950399999999998, 0), v100, z5, tool0;
	MoveL Offs(p0,290.3256,12.3232, 0), v100, z5, tool0;
	MoveL Offs(p0,290.4304,11.8208, 0), v100, z5, tool0;
	MoveL Offs(p0,290.2568,11.4456, 0), v100, z5, tool0;
	MoveL Offs(p0,289.8,11.2, 0), v100, z5, tool0;
	MoveL Offs(p0,283.4032000000001,9.304, 0), v100, z5, tool0;
	MoveL Offs(p0,276.5216000000001,7.8160000000000025, 0), v100, z5, tool0;
	MoveL Offs(p0,269.2584,6.735999999999999, 0), v100, z5, tool0;
	MoveL Offs(p0,261.71680000000003,6.064, 0), v100, z5, tool0;
	MoveL Offs(p0,254.0,5.8, 0), v100, z5, tool0;
	MoveL Offs(p0,246.21120000000002,5.944000000000001, 0), v100, z5, tool0;
	MoveL Offs(p0,238.4536,6.496, 0), v100, z5, tool0;
	MoveL Offs(p0,230.8304,7.456, 0), v100, z5, tool0;
	MoveL Offs(p0,223.44480000000004,8.824000000000002, 0), v100, z5, tool0;
	MoveL Offs(p0,216.4,10.6, 0), v100, z5, tool0;
	MoveL Offs(p0,211.15940000000006,12.286800000000003, 0), v100, z5, tool0;
	MoveL Offs(p0,206.0352000000001,14.206400000000002, 0), v100, z5, tool0;
	MoveL Offs(p0,201.08379999999997,16.3276, 0), v100, z5, tool0;
	MoveL Offs(p0,196.3616,18.619200000000003, 0), v100, z5, tool0;
	MoveL Offs(p0,191.925,21.05, 0), v100, z5, tool0;
	MoveL Offs(p0,187.8304,23.5888, 0), v100, z5, tool0;
	MoveL Offs(p0,184.13420000000002,26.204400000000003, 0), v100, z5, tool0;
	MoveL Offs(p0,180.89280000000002,28.865600000000008, 0), v100, z5, tool0;
	MoveL Offs(p0,178.16260000000003,31.541200000000003, 0), v100, z5, tool0;
	MoveL Offs(p0,176.0,34.2, 0), v100, z5, tool0;
	MoveL Offs(p0,171.8,39.8, 0), v100, z5, tool0;
	MoveL Offs(p0,176.8,43.2, 0), v100, z5, tool0;
	MoveL Offs(p0,179.6712,44.8502, 0), v100, z5, tool0;
	MoveL Offs(p0,182.77760000000006,46.32160000000001, 0), v100, z5, tool0;
	MoveL Offs(p0,186.1384,47.6154, 0), v100, z5, tool0;
	MoveL Offs(p0,189.77280000000002,48.732800000000005, 0), v100, z5, tool0;
	MoveL Offs(p0,193.7,49.675, 0), v100, z5, tool0;
	MoveL Offs(p0,197.93919999999997,50.443200000000004, 0), v100, z5, tool0;
	MoveL Offs(p0,202.5096,51.038599999999995, 0), v100, z5, tool0;
	MoveL Offs(p0,207.43040000000002,51.4624, 0), v100, z5, tool0;
	MoveL Offs(p0,212.7208,51.7158, 0), v100, z5, tool0;
	MoveL Offs(p0,218.4,51.8, 0), v100, z5, tool0;
	MoveL Offs(p0,222.2288,51.824200000000005, 0), v100, z5, tool0;
	MoveL Offs(p0,225.79840000000007,51.77760000000001, 0), v100, z5, tool0;
	MoveL Offs(p0,229.1136,51.66139999999999, 0), v100, z5, tool0;
	MoveL Offs(p0,232.17920000000004,51.476800000000004, 0), v100, z5, tool0;
	MoveL Offs(p0,235.0,51.225, 0), v100, z5, tool0;
	MoveL Offs(p0,237.5808,50.9072, 0), v100, z5, tool0;
	MoveL Offs(p0,239.9264,50.5246, 0), v100, z5, tool0;
	MoveL Offs(p0,242.04160000000002,50.0784, 0), v100, z5, tool0;
	MoveL Offs(p0,243.9312,49.5698, 0), v100, z5, tool0;
	MoveL Offs(p0,245.6,49.0, 0), v100, z5, tool0;
	MoveL Offs(p0,245.6,49.0, 0), v100, z5, tool0;
	MoveJ Offs(p0,594.0,604.6, 10), v100, z1, tool0;
	MoveL Offs(p0,593.9328000000003,601.7872000000002, 0), v100, z5, tool0;
	MoveL Offs(p0,593.8542,600.2097999999999, 0), v100, z5, tool0;
	MoveL Offs(p0,593.7504,598.5616000000001, 0), v100, z5, tool0;
	MoveL Offs(p0,593.625,596.875, 0), v100, z5, tool0;
	MoveL Offs(p0,593.4815999999998,595.1823999999999, 0), v100, z5, tool0;
	MoveL Offs(p0,593.3237999999999,593.5162, 0), v100, z5, tool0;
	MoveL Offs(p0,593.1552,591.9087999999999, 0), v100, z5, tool0;
	MoveL Offs(p0,592.9793999999999,590.3926, 0), v100, z5, tool0;
	MoveL Offs(p0,592.8,589.0, 0), v100, z5, tool0;
	MoveL Offs(p0,592.5320000000002,586.8856, 0), v100, z5, tool0;
	MoveL Offs(p0,592.3360000000001,585.2128000000001, 0), v100, z5, tool0;
	MoveL Offs(p0,592.224,583.9671999999999, 0), v100, z5, tool0;
	MoveL Offs(p0,592.2080000000001,583.1344, 0), v100, z5, tool0;
	MoveL Offs(p0,592.3,582.7, 0), v100, z5, tool0;
	MoveL Offs(p0,592.512,582.6496, 0), v100, z5, tool0;
	MoveL Offs(p0,592.856,582.9688, 0), v100, z5, tool0;
	MoveL Offs(p0,593.344,583.6432000000001, 0), v100, z5, tool0;
	MoveL Offs(p0,593.988,584.6584, 0), v100, z5, tool0;
	MoveL Offs(p0,594.8,586.0, 0), v100, z5, tool0;
	MoveL Offs(p0,595.7408000000001,588.0122, 0), v100, z5, tool0;
	MoveL Offs(p0,596.5184000000002,590.5776000000002, 0), v100, z5, tool0;
	MoveL Offs(p0,597.1256,593.5294, 0), v100, z5, tool0;
	MoveL Offs(p0,597.5552,596.7008000000001, 0), v100, z5, tool0;
	MoveL Offs(p0,597.8,599.925, 0), v100, z5, tool0;
	MoveL Offs(p0,597.8528,603.0351999999999, 0), v100, z5, tool0;
	MoveL Offs(p0,597.7064,605.8646, 0), v100, z5, tool0;
	MoveL Offs(p0,597.3536,608.2464, 0), v100, z5, tool0;
	MoveL Offs(p0,596.7872,610.0138, 0), v100, z5, tool0;
	MoveL Offs(p0,596.0,611.0, 0), v100, z5, tool0;
	MoveL Offs(p0,594.2052,608.1622, 0), v100, z5, tool0;
	MoveL Offs(p0,594.0928,607.1088, 0), v100, z5, tool0;
	MoveL Offs(p0,594.0236,605.9186, 0), v100, z5, tool0;
	MoveL Offs(p0,594.0,604.6, 0), v100, z5, tool0;
	MoveL Offs(p0,594.0,604.6, 0), v100, z5, tool0;
	MoveJ Offs(p0,592.8,543.2, 10), v100, z1, tool0;
	MoveL Offs(p0,590.5376000000002,541.9152000000001, 0), v100, z5, tool0;
	MoveL Offs(p0,589.1964,540.9788, 0), v100, z5, tool0;
	MoveL Offs(p0,587.7568,539.8816, 0), v100, z5, tool0;
	MoveL Offs(p0,586.25,538.65, 0), v100, z5, tool0;
	MoveL Offs(p0,584.7072000000001,537.3104, 0), v100, z5, tool0;
	MoveL Offs(p0,583.1596,535.8892, 0), v100, z5, tool0;
	MoveL Offs(p0,581.6384,534.4128000000001, 0), v100, z5, tool0;
	MoveL Offs(p0,580.1748,532.9076, 0), v100, z5, tool0;
	MoveL Offs(p0,578.8,531.4, 0), v100, z5, tool0;
	MoveL Offs(p0,575.5134,527.9412000000001, 0), v100, z5, tool0;
	MoveL Offs(p0,571.2992000000002,524.1296000000001, 0), v100, z5, tool0;
	MoveL Offs(p0,566.3457999999999,520.0924, 0), v100, z5, tool0;
	MoveL Offs(p0,560.8416,515.9568, 0), v100, z5, tool0;
	MoveL Offs(p0,554.975,511.85, 0), v100, z5, tool0;
	MoveL Offs(p0,548.9344,507.89919999999995, 0), v100, z5, tool0;
	MoveL Offs(p0,542.9082000000001,504.23159999999996, 0), v100, z5, tool0;
	MoveL Offs(p0,537.0848000000001,500.97440000000006, 0), v100, z5, tool0;
	MoveL Offs(p0,531.6526,498.25480000000005, 0), v100, z5, tool0;
	MoveL Offs(p0,526.8,496.2, 0), v100, z5, tool0;
	MoveL Offs(p0,522.9440000000002,494.8704000000001, 0), v100, z5, tool0;
	MoveL Offs(p0,520.7969999999999,494.2145999999999, 0), v100, z5, tool0;
	MoveL Offs(p0,518.5600000000001,493.5792, 0), v100, z5, tool0;
	MoveL Offs(p0,516.275,492.975, 0), v100, z5, tool0;
	MoveL Offs(p0,513.984,492.41279999999995, 0), v100, z5, tool0;
	MoveL Offs(p0,511.729,491.9034, 0), v100, z5, tool0;
	MoveL Offs(p0,509.552,491.45760000000007, 0), v100, z5, tool0;
	MoveL Offs(p0,507.49500000000006,491.0862, 0), v100, z5, tool0;
	MoveL Offs(p0,505.6,490.8, 0), v100, z5, tool0;
	MoveL Offs(p0,501.9408,490.2066000000001, 0), v100, z5, tool0;
	MoveL Offs(p0,498.6464000000002,489.38880000000006, 0), v100, z5, tool0;
	MoveL Offs(p0,495.7216,488.3502, 0), v100, z5, tool0;
	MoveL Offs(p0,493.17120000000006,487.09439999999995, 0), v100, z5, tool0;
	MoveL Offs(p0,491.0,485.625, 0), v100, z5, tool0;
	MoveL Offs(p0,489.21279999999996,483.9456, 0), v100, z5, tool0;
	MoveL Offs(p0,487.81440000000003,482.0598, 0), v100, z5, tool0;
	MoveL Offs(p0,486.80960000000005,479.9712000000001, 0), v100, z5, tool0;
	MoveL Offs(p0,486.20320000000004,477.68340000000006, 0), v100, z5, tool0;
	MoveL Offs(p0,486.0,475.2, 0), v100, z5, tool0;
	MoveL Offs(p0,487.0080000000001,471.4816000000002, 0), v100, z5, tool0;
	MoveL Offs(p0,488.37600000000003,468.7434, 0), v100, z5, tool0;
	MoveL Offs(p0,490.416,465.2768, 0), v100, z5, tool0;
	MoveL Offs(p0,493.2,460.975, 0), v100, z5, tool0;
	MoveL Offs(p0,496.8,455.7312, 0), v100, z5, tool0;
	MoveL Offs(p0,501.2879999999999,449.43859999999995, 0), v100, z5, tool0;
	MoveL Offs(p0,506.73600000000005,441.9904, 0), v100, z5, tool0;
	MoveL Offs(p0,513.216,433.2798000000001, 0), v100, z5, tool0;
	MoveL Offs(p0,520.8,423.2, 0), v100, z5, tool0;
	MoveL Offs(p0,530.1630000000001,410.71720000000005, 0), v100, z5, tool0;
	MoveL Offs(p0,537.8400000000003,400.3776000000001, 0), v100, z5, tool0;
	MoveL Offs(p0,544.173,391.62440000000004, 0), v100, z5, tool0;
	MoveL Offs(p0,549.5040000000001,383.9008, 0), v100, z5, tool0;
	MoveL Offs(p0,554.175,376.65, 0), v100, z5, tool0;
	MoveL Offs(p0,558.528,369.3152, 0), v100, z5, tool0;
	MoveL Offs(p0,562.905,361.33959999999996, 0), v100, z5, tool0;
	MoveL Offs(p0,567.648,352.1664, 0), v100, z5, tool0;
	MoveL Offs(p0,573.0989999999999,341.2388, 0), v100, z5, tool0;
	MoveL Offs(p0,579.6,328.0, 0), v100, z5, tool0;
	MoveL Offs(p0,583.5554,319.99100000000004, 0), v100, z5, tool0;
	MoveL Offs(p0,587.4592000000001,312.2400000000001, 0), v100, z5, tool0;
	MoveL Offs(p0,591.2478,304.861, 0), v100, z5, tool0;
	MoveL Offs(p0,594.8576,297.968, 0), v100, z5, tool0;
	MoveL Offs(p0,598.225,291.675, 0), v100, z5, tool0;
	MoveL Offs(p0,601.2864,286.096, 0), v100, z5, tool0;
	MoveL Offs(p0,603.9782,281.34499999999997, 0), v100, z5, tool0;
	MoveL Offs(p0,606.2368,277.536, 0), v100, z5, tool0;
	MoveL Offs(p0,607.9986,274.783, 0), v100, z5, tool0;
	MoveL Offs(p0,609.2,273.2, 0), v100, z5, tool0;
	MoveL Offs(p0,611.6896000000002,270.70560000000006, 0), v100, z5, tool0;
	MoveL Offs(p0,612.8054,269.81239999999997, 0), v100, z5, tool0;
	MoveL Offs(p0,613.9008,269.1328, 0), v100, z5, tool0;
	MoveL Offs(p0,615.025,268.65, 0), v100, z5, tool0;
	MoveL Offs(p0,616.2272,268.3472, 0), v100, z5, tool0;
	MoveL Offs(p0,617.5566,268.2076, 0), v100, z5, tool0;
	MoveL Offs(p0,619.0624,268.2144, 0), v100, z5, tool0;
	MoveL Offs(p0,620.7938,268.35080000000005, 0), v100, z5, tool0;
	MoveL Offs(p0,622.8,268.6, 0), v100, z5, tool0;
	MoveL Offs(p0,626.8472,269.62460000000004, 0), v100, z5, tool0;
	MoveL Offs(p0,632.8576000000002,271.8528000000001, 0), v100, z5, tool0;
	MoveL Offs(p0,640.4544,275.0962, 0), v100, z5, tool0;
	MoveL Offs(p0,649.2608000000001,279.16639999999995, 0), v100, z5, tool0;
	MoveL Offs(p0,658.9,283.875, 0), v100, z5, tool0;
	MoveL Offs(p0,668.9952,289.0336, 0), v100, z5, tool0;
	MoveL Offs(p0,679.1696,294.4538, 0), v100, z5, tool0;
	MoveL Offs(p0,689.0464000000001,299.9472, 0), v100, z5, tool0;
	MoveL Offs(p0,698.2488000000001,305.3254, 0), v100, z5, tool0;
	MoveL Offs(p0,706.4,310.4, 0), v100, z5, tool0;
	MoveL Offs(p0,712.2072000000001,314.26660000000004, 0), v100, z5, tool0;
	MoveL Offs(p0,716.9536000000003,317.66880000000003, 0), v100, z5, tool0;
	MoveL Offs(p0,720.7064,320.7302, 0), v100, z5, tool0;
	MoveL Offs(p0,723.5328000000001,323.5744, 0), v100, z5, tool0;
	MoveL Offs(p0,725.5,326.325, 0), v100, z5, tool0;
	MoveL Offs(p0,726.6752,329.1056, 0), v100, z5, tool0;
	MoveL Offs(p0,727.1256,332.0398, 0), v100, z5, tool0;
	MoveL Offs(p0,726.9184000000001,335.25120000000004, 0), v100, z5, tool0;
	MoveL Offs(p0,726.1208,338.8634, 0), v100, z5, tool0;
	MoveL Offs(p0,724.8,343.0, 0), v100, z5, tool0;
	MoveL Offs(p0,722.0754,350.14880000000005, 0), v100, z5, tool0;
	MoveL Offs(p0,718.2912000000002,358.8624000000001, 0), v100, z5, tool0;
	MoveL Offs(p0,713.5518,368.9416, 0), v100, z5, tool0;
	MoveL Offs(p0,707.9616,380.1872, 0), v100, z5, tool0;
	MoveL Offs(p0,701.625,392.4, 0), v100, z5, tool0;
	MoveL Offs(p0,694.6464,405.3808, 0), v100, z5, tool0;
	MoveL Offs(p0,687.1302,418.9304, 0), v100, z5, tool0;
	MoveL Offs(p0,679.1808000000001,432.8496000000001, 0), v100, z5, tool0;
	MoveL Offs(p0,670.9026,446.93919999999997, 0), v100, z5, tool0;
	MoveL Offs(p0,662.4,461.0, 0), v100, z5, tool0;
	MoveL Offs(p0,652.2412,477.59040000000005, 0), v100, z5, tool0;
	MoveL Offs(p0,643.3136000000002,492.03520000000015, 0), v100, z5, tool0;
	MoveL Offs(p0,635.5404,504.44479999999993, 0), v100, z5, tool0;
	MoveL Offs(p0,628.8448000000001,514.9296, 0), v100, z5, tool0;
	MoveL Offs(p0,623.15,523.6, 0), v100, z5, tool0;
	MoveL Offs(p0,618.3792000000001,530.5663999999999, 0), v100, z5, tool0;
	MoveL Offs(p0,614.4556,535.9392, 0), v100, z5, tool0;
	MoveL Offs(p0,611.3024,539.8288, 0), v100, z5, tool0;
	MoveL Offs(p0,608.8428,542.3456, 0), v100, z5, tool0;
	MoveL Offs(p0,607.0,543.6, 0), v100, z5, tool0;
	MoveL Offs(p0,603.8144000000001,545.0368000000001, 0), v100, z5, tool0;
	MoveL Offs(p0,602.5845999999999,545.4791999999999, 0), v100, z5, tool0;
	MoveL Offs(p0,601.4832,545.7344, 0), v100, z5, tool0;
	MoveL Offs(p0,600.425,545.8, 0), v100, z5, tool0;
	MoveL Offs(p0,599.3248,545.6736, 0), v100, z5, tool0;
	MoveL Offs(p0,598.0974,545.3528, 0), v100, z5, tool0;
	MoveL Offs(p0,596.6576000000001,544.8352000000001, 0), v100, z5, tool0;
	MoveL Offs(p0,594.9202,544.1184000000001, 0), v100, z5, tool0;
	MoveL Offs(p0,592.8,543.2, 0), v100, z5, tool0;
	MoveL Offs(p0,592.8,543.2, 0), v100, z5, tool0;
	MoveJ Offs(p0,606.0,538.0, 10), v100, z1, tool0;
	MoveL Offs(p0,608.7520000000002,535.6000000000001, 0), v100, z5, tool0;
	MoveL Offs(p0,609.933,533.7969999999999, 0), v100, z5, tool0;
	MoveL Offs(p0,610.9760000000001,531.6160000000001, 0), v100, z5, tool0;
	MoveL Offs(p0,611.875,529.075, 0), v100, z5, tool0;
	MoveL Offs(p0,612.624,526.192, 0), v100, z5, tool0;
	MoveL Offs(p0,613.217,522.985, 0), v100, z5, tool0;
	MoveL Offs(p0,613.6480000000001,519.4720000000001, 0), v100, z5, tool0;
	MoveL Offs(p0,613.9110000000001,515.671, 0), v100, z5, tool0;
	MoveL Offs(p0,614.0,511.6, 0), v100, z5, tool0;
	MoveL Offs(p0,613.8828000000001,507.2368, 0), v100, z5, tool0;
	MoveL Offs(p0,613.5184000000002,503.7424000000001, 0), v100, z5, tool0;
	MoveL Offs(p0,612.8876,501.10959999999994, 0), v100, z5, tool0;
	MoveL Offs(p0,611.9712000000001,499.33119999999997, 0), v100, z5, tool0;
	MoveL Offs(p0,610.75,498.4, 0), v100, z5, tool0;
	MoveL Offs(p0,609.2048,498.30879999999996, 0), v100, z5, tool0;
	MoveL Offs(p0,607.3164,499.05039999999997, 0), v100, z5, tool0;
	MoveL Offs(p0,605.0656000000001,500.61760000000004, 0), v100, z5, tool0;
	MoveL Offs(p0,602.4332,503.0032, 0), v100, z5, tool0;
	MoveL Offs(p0,599.4,506.2, 0), v100, z5, tool0;
	MoveL Offs(p0,596.5308000000001,509.5570000000001, 0), v100, z5, tool0;
	MoveL Offs(p0,594.0384000000003,512.6800000000001, 0), v100, z5, tool0;
	MoveL Offs(p0,591.9155999999999,515.587, 0), v100, z5, tool0;
	MoveL Offs(p0,590.1551999999999,518.296, 0), v100, z5, tool0;
	MoveL Offs(p0,588.75,520.825, 0), v100, z5, tool0;
	MoveL Offs(p0,587.6928,523.192, 0), v100, z5, tool0;
	MoveL Offs(p0,586.9764,525.415, 0), v100, z5, tool0;
	MoveL Offs(p0,586.5936,527.5120000000001, 0), v100, z5, tool0;
	MoveL Offs(p0,586.5372,529.501, 0), v100, z5, tool0;
	MoveL Offs(p0,586.8,531.4, 0), v100, z5, tool0;
	MoveL Offs(p0,588.7776000000001,535.1584000000001, 0), v100, z5, tool0;
	MoveL Offs(p0,590.3424,536.6686, 0), v100, z5, tool0;
	MoveL Offs(p0,592.2048000000001,537.8992000000001, 0), v100, z5, tool0;
	MoveL Offs(p0,594.3,538.825, 0), v100, z5, tool0;
	MoveL Offs(p0,596.5631999999999,539.4208000000001, 0), v100, z5, tool0;
	MoveL Offs(p0,598.9296,539.6614, 0), v100, z5, tool0;
	MoveL Offs(p0,601.3344000000001,539.5216, 0), v100, z5, tool0;
	MoveL Offs(p0,603.7128,538.9762000000001, 0), v100, z5, tool0;
	MoveL Offs(p0,606.0,538.0, 0), v100, z5, tool0;
	MoveL Offs(p0,606.0,538.0, 0), v100, z5, tool0;
	MoveJ Offs(p0,513.6,481.8, 10), v100, z1, tool0;
	MoveL Offs(p0,516.5792000000001,477.48960000000017, 0), v100, z5, tool0;
	MoveL Offs(p0,518.2188,474.42539999999997, 0), v100, z5, tool0;
	MoveL Offs(p0,519.8656,470.9808, 0), v100, z5, tool0;
	MoveL Offs(p0,521.45,467.325, 0), v100, z5, tool0;
	MoveL Offs(p0,522.9024000000001,463.6272, 0), v100, z5, tool0;
	MoveL Offs(p0,524.1532,460.0566, 0), v100, z5, tool0;
	MoveL Offs(p0,525.1328000000001,456.78240000000005, 0), v100, z5, tool0;
	MoveL Offs(p0,525.7716,453.97380000000004, 0), v100, z5, tool0;
	MoveL Offs(p0,526.0,451.8, 0), v100, z5, tool0;
	MoveL Offs(p0,525.5074000000001,449.6474, 0), v100, z5, tool0;
	MoveL Offs(p0,524.1232000000001,448.4272000000001, 0), v100, z5, tool0;
	MoveL Offs(p0,521.9878,448.07579999999996, 0), v100, z5, tool0;
	MoveL Offs(p0,519.2416000000001,448.5296, 0), v100, z5, tool0;
	MoveL Offs(p0,516.025,449.725, 0), v100, z5, tool0;
	MoveL Offs(p0,512.4784,451.5984, 0), v100, z5, tool0;
	MoveL Offs(p0,508.74219999999997,454.0862, 0), v100, z5, tool0;
	MoveL Offs(p0,504.9568000000001,457.12480000000005, 0), v100, z5, tool0;
	MoveL Offs(p0,501.2626,460.65060000000005, 0), v100, z5, tool0;
	MoveL Offs(p0,497.8,464.6, 0), v100, z5, tool0;
	MoveL Offs(p0,496.40740000000005,466.6594000000001, 0), v100, z5, tool0;
	MoveL Offs(p0,495.34720000000016,468.7392000000001, 0), v100, z5, tool0;
	MoveL Offs(p0,494.61580000000004,470.81179999999995, 0), v100, z5, tool0;
	MoveL Offs(p0,494.20959999999997,472.8496000000001, 0), v100, z5, tool0;
	MoveL Offs(p0,494.125,474.825, 0), v100, z5, tool0;
	MoveL Offs(p0,494.35839999999996,476.71039999999994, 0), v100, z5, tool0;
	MoveL Offs(p0,494.9062,478.4781999999999, 0), v100, z5, tool0;
	MoveL Offs(p0,495.7648000000001,480.10080000000005, 0), v100, z5, tool0;
	MoveL Offs(p0,496.9306,481.55060000000003, 0), v100, z5, tool0;
	MoveL Offs(p0,498.4,482.8, 0), v100, z5, tool0;
	MoveL Offs(p0,501.84320000000014,484.8656000000002, 0), v100, z5, tool0;
	MoveL Offs(p0,503.4598,485.46940000000006, 0), v100, z5, tool0;
	MoveL Offs(p0,505.01759999999996,485.7888, 0), v100, z5, tool0;
	MoveL Offs(p0,506.525,485.825, 0), v100, z5, tool0;
	MoveL Offs(p0,507.9904,485.57919999999996, 0), v100, z5, tool0;
	MoveL Offs(p0,509.4222,485.0526, 0), v100, z5, tool0;
	MoveL Offs(p0,510.82880000000006,484.2464000000001, 0), v100, z5, tool0;
	MoveL Offs(p0,512.2186,483.1618, 0), v100, z5, tool0;
	MoveL Offs(p0,513.6,481.8, 0), v100, z5, tool0;
	MoveL Offs(p0,513.6,481.8, 0), v100, z5, tool0;
	MoveJ Offs(p0,655.8,448.6, 10), v100, z1, tool0;
	MoveL Offs(p0,658.7956,445.40780000000007, 0), v100, z5, tool0;
	MoveL Offs(p0,663.2288000000001,439.4544000000002, 0), v100, z5, tool0;
	MoveL Offs(p0,668.7492,431.3146, 0), v100, z5, tool0;
	MoveL Offs(p0,675.0064,421.56320000000005, 0), v100, z5, tool0;
	MoveL Offs(p0,681.65,410.775, 0), v100, z5, tool0;
	MoveL Offs(p0,688.3296,399.5248, 0), v100, z5, tool0;
	MoveL Offs(p0,694.6948,388.38739999999996, 0), v100, z5, tool0;
	MoveL Offs(p0,700.3952,377.93760000000003, 0), v100, z5, tool0;
	MoveL Offs(p0,705.0804,368.7502, 0), v100, z5, tool0;
	MoveL Offs(p0,708.4,361.4, 0), v100, z5, tool0;
	MoveL Offs(p0,709.1685999999999,359.24719999999996, 0), v100, z5, tool0;
	MoveL Offs(p0,709.1712,358.9264, 0), v100, z5, tool0;
	MoveL Offs(p0,709.025,358.8, 0), v100, z5, tool0;
	MoveL Offs(p0,708.7167999999999,358.8656, 0), v100, z5, tool0;
	MoveL Offs(p0,708.2334,359.1208, 0), v100, z5, tool0;
	MoveL Offs(p0,705.6,361.0, 0), v100, z5, tool0;
	MoveL Offs(p0,702.2368000000002,362.82240000000013, 0), v100, z5, tool0;
	MoveL Offs(p0,700.6661999999999,363.3886, 0), v100, z5, tool0;
	MoveL Offs(p0,699.1904000000001,363.7232, 0), v100, z5, tool0;
	MoveL Offs(p0,697.825,363.825, 0), v100, z5, tool0;
	MoveL Offs(p0,696.5856000000001,363.6928, 0), v100, z5, tool0;
	MoveL Offs(p0,695.4878,363.3254, 0), v100, z5, tool0;
	MoveL Offs(p0,694.5472000000001,362.7216, 0), v100, z5, tool0;
	MoveL Offs(p0,693.7794000000001,361.8802, 0), v100, z5, tool0;
	MoveL Offs(p0,693.2,360.8, 0), v100, z5, tool0;
	MoveL Offs(p0,692.6346000000001,358.59720000000004, 0), v100, z5, tool0;
	MoveL Offs(p0,692.2528000000001,355.5856000000001, 0), v100, z5, tool0;
	MoveL Offs(p0,692.0462,351.9404, 0), v100, z5, tool0;
	MoveL Offs(p0,692.0064000000001,347.8368, 0), v100, z5, tool0;
	MoveL Offs(p0,692.125,343.45, 0), v100, z5, tool0;
	MoveL Offs(p0,692.3936000000001,338.9552, 0), v100, z5, tool0;
	MoveL Offs(p0,692.8037999999999,334.5276, 0), v100, z5, tool0;
	MoveL Offs(p0,693.3472,330.3424, 0), v100, z5, tool0;
	MoveL Offs(p0,694.0154,326.5748, 0), v100, z5, tool0;
	MoveL Offs(p0,694.8,323.4, 0), v100, z5, tool0;
	MoveL Offs(p0,697.6,314.0, 0), v100, z5, tool0;
	MoveL Offs(p0,688.0,308.2, 0), v100, z5, tool0;
	MoveL Offs(p0,683.9328000000003,305.77760000000006, 0), v100, z5, tool0;
	MoveL Offs(p0,681.2841999999999,304.24539999999996, 0), v100, z5, tool0;
	MoveL Offs(p0,678.3104000000001,302.5488, 0), v100, z5, tool0;
	MoveL Offs(p0,675.075,300.725, 0), v100, z5, tool0;
	MoveL Offs(p0,671.6416,298.8112, 0), v100, z5, tool0;
	MoveL Offs(p0,668.0737999999999,296.8446, 0), v100, z5, tool0;
	MoveL Offs(p0,664.4352000000001,294.86240000000004, 0), v100, z5, tool0;
	MoveL Offs(p0,660.7894,292.9018, 0), v100, z5, tool0;
	MoveL Offs(p0,657.2,291.0, 0), v100, z5, tool0;
	MoveL Offs(p0,652.4754,288.4702000000001, 0), v100, z5, tool0;
	MoveL Offs(p0,648.4672000000003,286.38560000000007, 0), v100, z5, tool0;
	MoveL Offs(p0,645.1238,284.72339999999997, 0), v100, z5, tool0;
	MoveL Offs(p0,642.3936000000001,283.4608, 0), v100, z5, tool0;
	MoveL Offs(p0,640.225,282.575, 0), v100, z5, tool0;
	MoveL Offs(p0,638.5663999999999,282.04319999999996, 0), v100, z5, tool0;
	MoveL Offs(p0,637.3662,281.84260000000006, 0), v100, z5, tool0;
	MoveL Offs(p0,636.5728000000001,281.9504, 0), v100, z5, tool0;
	MoveL Offs(p0,636.1346000000001,282.3438, 0), v100, z5, tool0;
	MoveL Offs(p0,636.0,283.0, 0), v100, z5, tool0;
	MoveL Offs(p0,635.1568000000001,286.92320000000007, 0), v100, z5, tool0;
	MoveL Offs(p0,634.1532,289.1488, 0), v100, z5, tool0;
	MoveL Offs(p0,632.8064000000002,291.48960000000005, 0), v100, z5, tool0;
	MoveL Offs(p0,631.15,293.9, 0), v100, z5, tool0;
	MoveL Offs(p0,629.2176,296.3344, 0), v100, z5, tool0;
	MoveL Offs(p0,627.0427999999999,298.74719999999996, 0), v100, z5, tool0;
	MoveL Offs(p0,624.6592,301.0928, 0), v100, z5, tool0;
	MoveL Offs(p0,622.1004,303.3256, 0), v100, z5, tool0;
	MoveL Offs(p0,619.4,305.4, 0), v100, z5, tool0;
	MoveL Offs(p0,616.3536000000001,307.52340000000004, 0), v100, z5, tool0;
	MoveL Offs(p0,613.4608000000002,309.3312000000001, 0), v100, z5, tool0;
	MoveL Offs(p0,610.7312000000001,310.81980000000004, 0), v100, z5, tool0;
	MoveL Offs(p0,608.1744,311.98560000000003, 0), v100, z5, tool0;
	MoveL Offs(p0,605.8,312.825, 0), v100, z5, tool0;
	MoveL Offs(p0,603.6175999999999,313.3344, 0), v100, z5, tool0;
	MoveL Offs(p0,601.6368,313.5102, 0), v100, z5, tool0;
	MoveL Offs(p0,599.8672,313.34880000000004, 0), v100, z5, tool0;
	MoveL Offs(p0,598.3183999999999,312.8466, 0), v100, z5, tool0;
	MoveL Offs(p0,597.0,312.0, 0), v100, z5, tool0;
	MoveL Offs(p0,594.786,311.7389999999999, 0), v100, z5, tool0;
	MoveL Offs(p0,593.9280000000001,312.48, 0), v100, z5, tool0;
	MoveL Offs(p0,592.95,313.725, 0), v100, z5, tool0;
	MoveL Offs(p0,591.816,315.528, 0), v100, z5, tool0;
	MoveL Offs(p0,590.49,317.94300000000004, 0), v100, z5, tool0;
	MoveL Offs(p0,588.936,321.02400000000006, 0), v100, z5, tool0;
	MoveL Offs(p0,587.118,324.82500000000005, 0), v100, z5, tool0;
	MoveL Offs(p0,585.0,329.4, 0), v100, z5, tool0;
	MoveL Offs(p0,578.9968,342.6154, 0), v100, z5, tool0;
	MoveL Offs(p0,573.9344000000001,354.48320000000007, 0), v100, z5, tool0;
	MoveL Offs(p0,569.7936,365.0958, 0), v100, z5, tool0;
	MoveL Offs(p0,566.5552,374.54560000000004, 0), v100, z5, tool0;
	MoveL Offs(p0,564.2,382.925, 0), v100, z5, tool0;
	MoveL Offs(p0,562.7088,390.3264, 0), v100, z5, tool0;
	MoveL Offs(p0,562.0624,396.8422, 0), v100, z5, tool0;
	MoveL Offs(p0,562.2416000000001,402.5648, 0), v100, z5, tool0;
	MoveL Offs(p0,563.2272,407.5866, 0), v100, z5, tool0;
	MoveL Offs(p0,565.0,412.0, 0), v100, z5, tool0;
	MoveL Offs(p0,566.4326000000001,414.1078000000001, 0), v100, z5, tool0;
	MoveL Offs(p0,568.5888000000002,416.4064, 0), v100, z5, tool0;
	MoveL Offs(p0,571.3162,418.79859999999996, 0), v100, z5, tool0;
	MoveL Offs(p0,574.4624000000001,421.1872, 0), v100, z5, tool0;
	MoveL Offs(p0,577.875,423.475, 0), v100, z5, tool0;
	MoveL Offs(p0,581.4015999999999,425.5648, 0), v100, z5, tool0;
	MoveL Offs(p0,584.8898,427.3594, 0), v100, z5, tool0;
	MoveL Offs(p0,588.1872000000001,428.7616, 0), v100, z5, tool0;
	MoveL Offs(p0,591.1414000000001,429.67420000000004, 0), v100, z5, tool0;
	MoveL Offs(p0,593.6,430.0, 0), v100, z5, tool0;
	MoveL Offs(p0,596.5447999999999,430.79920000000004, 0), v100, z5, tool0;
	MoveL Offs(p0,597.7376,431.3824000000001, 0), v100, z5, tool0;
	MoveL Offs(p0,599.0,432.1, 0), v100, z5, tool0;
	MoveL Offs(p0,600.3104,432.93760000000003, 0), v100, z5, tool0;
	MoveL Offs(p0,601.6472,433.8808, 0), v100, z5, tool0;
	MoveL Offs(p0,602.9888000000001,434.9152, 0), v100, z5, tool0;
	MoveL Offs(p0,604.3136000000001,436.0264, 0), v100, z5, tool0;
	MoveL Offs(p0,605.6,437.2, 0), v100, z5, tool0;
	MoveL Offs(p0,610.5966000000001,441.6070000000001, 0), v100, z5, tool0;
	MoveL Offs(p0,615.8128000000003,445.33600000000007, 0), v100, z5, tool0;
	MoveL Offs(p0,621.1682,448.36899999999997, 0), v100, z5, tool0;
	MoveL Offs(p0,626.5824,450.688, 0), v100, z5, tool0;
	MoveL Offs(p0,631.975,452.275, 0), v100, z5, tool0;
	MoveL Offs(p0,637.2656,453.11199999999997, 0), v100, z5, tool0;
	MoveL Offs(p0,642.3738,453.1809999999999, 0), v100, z5, tool0;
	MoveL Offs(p0,647.2192000000001,452.46400000000006, 0), v100, z5, tool0;
	MoveL Offs(p0,651.7214,450.94300000000004, 0), v100, z5, tool0;
	MoveL Offs(p0,655.8,448.6, 0), v100, z5, tool0;
	MoveL Offs(p0,655.8,448.6, 0), v100, z5, tool0;
	MoveJ Offs(p0,710.4,350.0, 10), v100, z1, tool0;
	MoveL Offs(p0,712.8032000000002,347.15360000000015, 0), v100, z5, tool0;
	MoveL Offs(p0,713.8937999999999,345.7034, 0), v100, z5, tool0;
	MoveL Offs(p0,714.8896000000001,344.26880000000006, 0), v100, z5, tool0;
	MoveL Offs(p0,715.775,342.875, 0), v100, z5, tool0;
	MoveL Offs(p0,716.5343999999999,341.5472, 0), v100, z5, tool0;
	MoveL Offs(p0,717.1522,340.31059999999997, 0), v100, z5, tool0;
	MoveL Offs(p0,717.6128000000001,339.19040000000007, 0), v100, z5, tool0;
	MoveL Offs(p0,717.9005999999999,338.2118, 0), v100, z5, tool0;
	MoveL Offs(p0,718.0,337.4, 0), v100, z5, tool0;
	MoveL Offs(p0,717.4608000000002,333.8512000000001, 0), v100, z5, tool0;
	MoveL Offs(p0,716.8281999999999,332.0828, 0), v100, z5, tool0;
	MoveL Offs(p0,715.9904000000001,330.36960000000005, 0), v100, z5, tool0;
	MoveL Offs(p0,714.975,328.75, 0), v100, z5, tool0;
	MoveL Offs(p0,713.8095999999998,327.26239999999996, 0), v100, z5, tool0;
	MoveL Offs(p0,712.5217999999999,325.9452, 0), v100, z5, tool0;
	MoveL Offs(p0,711.1392000000001,324.83680000000004, 0), v100, z5, tool0;
	MoveL Offs(p0,709.6894,323.97560000000004, 0), v100, z5, tool0;
	MoveL Offs(p0,708.2,323.4, 0), v100, z5, tool0;
	MoveL Offs(p0,704.5184000000002,323.1056000000001, 0), v100, z5, tool0;
	MoveL Offs(p0,702.9656,323.5674, 0), v100, z5, tool0;
	MoveL Offs(p0,701.5952,324.45279999999997, 0), v100, z5, tool0;
	MoveL Offs(p0,700.4,325.775, 0), v100, z5, tool0;
	MoveL Offs(p0,699.3728,327.5472, 0), v100, z5, tool0;
	MoveL Offs(p0,698.5064,329.7826, 0), v100, z5, tool0;
	MoveL Offs(p0,697.7936000000001,332.49440000000004, 0), v100, z5, tool0;
	MoveL Offs(p0,697.2272,335.6958, 0), v100, z5, tool0;
	MoveL Offs(p0,696.8,339.4, 0), v100, z5, tool0;
	MoveL Offs(p0,696.3114000000002,345.09680000000003, 0), v100, z5, tool0;
	MoveL Offs(p0,696.1792000000003,349.7184000000001, 0), v100, z5, tool0;
	MoveL Offs(p0,696.4237999999999,353.28159999999997, 0), v100, z5, tool0;
	MoveL Offs(p0,697.0656,355.8032, 0), v100, z5, tool0;
	MoveL Offs(p0,698.125,357.3, 0), v100, z5, tool0;
	MoveL Offs(p0,699.6224,357.78880000000004, 0), v100, z5, tool0;
	MoveL Offs(p0,701.5781999999999,357.28639999999996, 0), v100, z5, tool0;
	MoveL Offs(p0,704.0128000000001,355.80960000000005, 0), v100, z5, tool0;
	MoveL Offs(p0,706.9466,353.37520000000006, 0), v100, z5, tool0;
	MoveL Offs(p0,710.4,350.0, 0), v100, z5, tool0;
	MoveL Offs(p0,710.4,350.0, 0), v100, z5, tool0;
	MoveJ Offs(p0,612.0,304.6, 10), v100, z1, tool0;
	MoveL Offs(p0,614.7322000000001,302.7142, 0), v100, z5, tool0;
	MoveL Offs(p0,617.2736000000002,300.7936000000001, 0), v100, z5, tool0;
	MoveL Offs(p0,619.6014,298.86339999999996, 0), v100, z5, tool0;
	MoveL Offs(p0,621.6928,296.9488, 0), v100, z5, tool0;
	MoveL Offs(p0,623.525,295.075, 0), v100, z5, tool0;
	MoveL Offs(p0,625.0752,293.2672, 0), v100, z5, tool0;
	MoveL Offs(p0,626.3206,291.55060000000003, 0), v100, z5, tool0;
	MoveL Offs(p0,627.2384,289.95040000000006, 0), v100, z5, tool0;
	MoveL Offs(p0,627.8058000000001,288.49179999999996, 0), v100, z5, tool0;
	MoveL Offs(p0,628.0,287.2, 0), v100, z5, tool0;
	MoveL Offs(p0,627.3808000000001,284.1152000000001, 0), v100, z5, tool0;
	MoveL Offs(p0,626.6662,282.5758, 0), v100, z5, tool0;
	MoveL Offs(p0,625.7344,281.0976, 0), v100, z5, tool0;
	MoveL Offs(p0,624.625,279.725, 0), v100, z5, tool0;
	MoveL Offs(p0,623.3776,278.50239999999997, 0), v100, z5, tool0;
	MoveL Offs(p0,622.0318,277.4742, 0), v100, z5, tool0;
	MoveL Offs(p0,620.6272000000001,276.6848, 0), v100, z5, tool0;
	MoveL Offs(p0,619.2034000000001,276.1786, 0), v100, z5, tool0;
	MoveL Offs(p0,617.8,276.0, 0), v100, z5, tool0;
	MoveL Offs(p0,614.5632000000002,277.1792000000001, 0), v100, z5, tool0;
	MoveL Offs(p0,612.7618,278.54879999999997, 0), v100, z5, tool0;
	MoveL Offs(p0,610.9136000000001,280.3456, 0), v100, z5, tool0;
	MoveL Offs(p0,609.075,282.5, 0), v100, z5, tool0;
	MoveL Offs(p0,607.3024,284.9424, 0), v100, z5, tool0;
	MoveL Offs(p0,605.6522,287.6032, 0), v100, z5, tool0;
	MoveL Offs(p0,604.1808000000001,290.4128, 0), v100, z5, tool0;
	MoveL Offs(p0,602.9446,293.3016, 0), v100, z5, tool0;
	MoveL Offs(p0,602.0,296.2, 0), v100, z5, tool0;
	MoveL Offs(p0,601.2432000000001,299.5294, 0), v100, z5, tool0;
	MoveL Offs(p0,600.8896000000002,302.31520000000006, 0), v100, z5, tool0;
	MoveL Offs(p0,600.9343999999999,304.5538, 0), v100, z5, tool0;
	MoveL Offs(p0,601.3728000000001,306.2416, 0), v100, z5, tool0;
	MoveL Offs(p0,602.2,307.375, 0), v100, z5, tool0;
	MoveL Offs(p0,603.4112,307.9504, 0), v100, z5, tool0;
	MoveL Offs(p0,605.0015999999999,307.9642, 0), v100, z5, tool0;
	MoveL Offs(p0,606.9664,307.41280000000006, 0), v100, z5, tool0;
	MoveL Offs(p0,609.3008,306.2926, 0), v100, z5, tool0;
	MoveL Offs(p0,612.0,304.6, 0), v100, z5, tool0;
	MoveL Offs(p0,612.0,304.6, 0), v100, z5, tool0;
	MoveJ Offs(p0,544.2,556.2, 10), v100, z1, tool0;
	MoveL Offs(p0,542.0288000000003,553.5264000000001, 0), v100, z5, tool0;
	MoveL Offs(p0,541.2191999999999,552.1446, 0), v100, z5, tool0;
	MoveL Offs(p0,540.6064,550.7952000000001, 0), v100, z5, tool0;
	MoveL Offs(p0,540.2,549.525, 0), v100, z5, tool0;
	MoveL Offs(p0,540.0096000000001,548.3808, 0), v100, z5, tool0;
	MoveL Offs(p0,540.0448,547.4094, 0), v100, z5, tool0;
	MoveL Offs(p0,540.3152,546.6576000000001, 0), v100, z5, tool0;
	MoveL Offs(p0,540.8304,546.1722, 0), v100, z5, tool0;
	MoveL Offs(p0,541.6,546.0, 0), v100, z5, tool0;
	MoveL Offs(p0,544.2,547.45, 0), v100, z5, tool0;
	MoveL Offs(p0,544.912,548.0304, 0), v100, z5, tool0;
	MoveL Offs(p0,545.6600000000001,548.6852, 0), v100, z5, tool0;
	MoveL Offs(p0,546.432,549.4048, 0), v100, z5, tool0;
	MoveL Offs(p0,547.216,550.1796, 0), v100, z5, tool0;
	MoveL Offs(p0,548.0,551.0, 0), v100, z5, tool0;
	MoveL Offs(p0,550.3634,553.8403999999999, 0), v100, z5, tool0;
	MoveL Offs(p0,550.8448000000001,554.6288000000002, 0), v100, z5, tool0;
	MoveL Offs(p0,551.175,555.35, 0), v100, z5, tool0;
	MoveL Offs(p0,551.3552,556.0112, 0), v100, z5, tool0;
	MoveL Offs(p0,551.3866,556.6196, 0), v100, z5, tool0;
	MoveL Offs(p0,551.2704,557.1824, 0), v100, z5, tool0;
	MoveL Offs(p0,551.0078000000001,557.7068, 0), v100, z5, tool0;
	MoveL Offs(p0,550.6,558.2, 0), v100, z5, tool0;
	MoveL Offs(p0,548.5200000000001,559.0512, 0), v100, z5, tool0;
	MoveL Offs(p0,547.925,558.925, 0), v100, z5, tool0;
	MoveL Offs(p0,547.288,558.6608, 0), v100, z5, tool0;
	MoveL Offs(p0,546.603,558.2574000000001, 0), v100, z5, tool0;
	MoveL Offs(p0,545.864,557.7136, 0), v100, z5, tool0;
	MoveL Offs(p0,545.0649999999999,557.0282, 0), v100, z5, tool0;
	MoveL Offs(p0,544.2,556.2, 0), v100, z5, tool0;
	MoveL Offs(p0,544.2,556.2, 0), v100, z5, tool0;
	MoveJ Offs(p0,495.6,529.8, 10), v100, z1, tool0;
	MoveL Offs(p0,492.93600000000004,527.145, 0), v100, z5, tool0;
	MoveL Offs(p0,492.416,526.104, 0), v100, z5, tool0;
	MoveL Offs(p0,492.1,525.075, 0), v100, z5, tool0;
	MoveL Offs(p0,492.0,524.112, 0), v100, z5, tool0;
	MoveL Offs(p0,492.128,523.269, 0), v100, z5, tool0;
	MoveL Offs(p0,492.4960000000001,522.6, 0), v100, z5, tool0;
	MoveL Offs(p0,493.1160000000001,522.159, 0), v100, z5, tool0;
	MoveL Offs(p0,494.0,522.0, 0), v100, z5, tool0;
	MoveL Offs(p0,496.496,522.6080000000001, 0), v100, z5, tool0;
	MoveL Offs(p0,497.375,522.925, 0), v100, z5, tool0;
	MoveL Offs(p0,498.32000000000005,523.296, 0), v100, z5, tool0;
	MoveL Offs(p0,499.313,523.7149999999999, 0), v100, z5, tool0;
	MoveL Offs(p0,500.33600000000007,524.176, 0), v100, z5, tool0;
	MoveL Offs(p0,501.3710000000001,524.673, 0), v100, z5, tool0;
	MoveL Offs(p0,502.4,525.2, 0), v100, z5, tool0;
	MoveL Offs(p0,504.80800000000016,526.5072000000002, 0), v100, z5, tool0;
	MoveL Offs(p0,505.6669999999999,527.0737999999999, 0), v100, z5, tool0;
	MoveL Offs(p0,506.3040000000001,527.5936, 0), v100, z5, tool0;
	MoveL Offs(p0,506.725,528.075, 0), v100, z5, tool0;
	MoveL Offs(p0,506.936,528.5264, 0), v100, z5, tool0;
	MoveL Offs(p0,506.94300000000004,528.9562, 0), v100, z5, tool0;
	MoveL Offs(p0,506.75200000000007,529.3728000000001, 0), v100, z5, tool0;
	MoveL Offs(p0,506.369,529.7846000000001, 0), v100, z5, tool0;
	MoveL Offs(p0,505.8,530.2, 0), v100, z5, tool0;
	MoveL Offs(p0,503.7600000000001,531.2528000000001, 0), v100, z5, tool0;
	MoveL Offs(p0,502.803,531.5752, 0), v100, z5, tool0;
	MoveL Offs(p0,501.86400000000003,531.7583999999999, 0), v100, z5, tool0;
	MoveL Offs(p0,500.925,531.8, 0), v100, z5, tool0;
	MoveL Offs(p0,499.968,531.6976, 0), v100, z5, tool0;
	MoveL Offs(p0,498.975,531.4487999999999, 0), v100, z5, tool0;
	MoveL Offs(p0,497.92800000000005,531.0512000000001, 0), v100, z5, tool0;
	MoveL Offs(p0,496.809,530.5024000000001, 0), v100, z5, tool0;
	MoveL Offs(p0,495.6,529.8, 0), v100, z5, tool0;
	MoveL Offs(p0,495.6,529.8, 0), v100, z5, tool0;
	MoveJ Offs(p0,435.8,512.0, 10), v100, z1, tool0;
	MoveL Offs(p0,439.5952000000001,508.71200000000016, 0), v100, z5, tool0;
	MoveL Offs(p0,441.2468,507.45500000000004, 0), v100, z5, tool0;
	MoveL Offs(p0,442.78560000000004,506.4320000000001, 0), v100, z5, tool0;
	MoveL Offs(p0,444.25,505.625, 0), v100, z5, tool0;
	MoveL Offs(p0,445.67840000000007,505.01599999999996, 0), v100, z5, tool0;
	MoveL Offs(p0,447.10920000000004,504.587, 0), v100, z5, tool0;
	MoveL Offs(p0,448.58080000000007,504.32000000000005, 0), v100, z5, tool0;
	MoveL Offs(p0,450.1316,504.197, 0), v100, z5, tool0;
	MoveL Offs(p0,451.8,504.2, 0), v100, z5, tool0;
	MoveL Offs(p0,459.0,504.4, 0), v100, z5, tool0;
	MoveL Offs(p0,453.0,506.4, 0), v100, z5, tool0;
	MoveL Offs(p0,450.71360000000016,507.3840000000002, 0), v100, z5, tool0;
	MoveL Offs(p0,449.3424,508.047, 0), v100, z5, tool0;
	MoveL Offs(p0,447.86080000000004,508.8, 0), v100, z5, tool0;
	MoveL Offs(p0,446.3,509.625, 0), v100, z5, tool0;
	MoveL Offs(p0,444.69120000000004,510.504, 0), v100, z5, tool0;
	MoveL Offs(p0,443.0656,511.419, 0), v100, z5, tool0;
	MoveL Offs(p0,441.45439999999996,512.3520000000001, 0), v100, z5, tool0;
	MoveL Offs(p0,439.88880000000006,513.2850000000001, 0), v100, z5, tool0;
	MoveL Offs(p0,438.4,514.2, 0), v100, z5, tool0;
	MoveL Offs(p0,435.1304000000001,516.3308000000001, 0), v100, z5, tool0;
	MoveL Offs(p0,432.5232000000001,517.9264000000001, 0), v100, z5, tool0;
	MoveL Offs(p0,430.5808,518.9916, 0), v100, z5, tool0;
	MoveL Offs(p0,429.3056,519.5312000000001, 0), v100, z5, tool0;
	MoveL Offs(p0,428.7,519.55, 0), v100, z5, tool0;
	MoveL Offs(p0,428.7664,519.0528, 0), v100, z5, tool0;
	MoveL Offs(p0,429.5072,518.0444, 0), v100, z5, tool0;
	MoveL Offs(p0,430.92480000000006,516.5296000000001, 0), v100, z5, tool0;
	MoveL Offs(p0,433.02160000000003,514.5132000000001, 0), v100, z5, tool0;
	MoveL Offs(p0,435.8,512.0, 0), v100, z5, tool0;
	MoveL Offs(p0,435.8,512.0, 0), v100, z5, tool0;
	ENDPROC
ENDMODULE
